// TwinCAT 3 PLC project TcoDrivesBeckhoff
// Title: TcoDrivesBeckhoff
// Company: Vortex.Library
// Author: TcOpenGroup
// ProjectVersion: 0.6.0.913
// ProgramVersion: 3.1.4024.12
// libraries:
//   Tc2_MC2, * (Beckhoff Automation GmbH)
//   Tc2_MC2_Drive, * (Beckhoff Automation GmbH)
//   Tc2_Standard, * (Beckhoff Automation GmbH)
//   Tc2_System, * (Beckhoff Automation GmbH)
//   Tc3_Module, * (Beckhoff Automation GmbH)
//   TcoCore, 0.6.0.913 (Vortex.Library)
// project tree:
//   DUTs/ eAxisParameter.TcDUT, eAxisEncoderReferenceSystem.TcDUT, eDirection.TcDUT, eAxisStates.TcDUT, eEncoderReferenceMode.TcDUT, eHomingMode.TcDUT, ePowerOverride.TcDUT, eSetPositionMode.TcDUT, eJogMode.TcDUT, TcoAxisOpModes.TcDUT, TcoAxisRef.TcPOU, TcoAxisStatus.TcDUT, TcoAxisConfig.TcDUT
//   / PlcTask.TcTTO (not stored)
//   POUs/Conversions/ Tc2MC2_TO_Tco_AxisStates.TcPOU, LREAL_TO_Tco_AxisEncoderReferenceSystem.TcPOU, Tc2MC2_TO_Tco_SetPositionMode.TcPOU, Tc2MC2_TO_Tco_JogMode.TcPOU, Tco_TO_Tc2MC2_SetPositionMode.TcPOU, Tco_TO_Tc2MC2_Direction.TcPOU, Tc2MC2_TO_Tco_Direction.TcPOU, Tco_TO_Tc2MC2_HomingMode.TcPOU, Tco_TO_Tc2MC2_EncRefMode.TcPOU, Tc2MC2_TO_Tco_EncRefMode.TcPOU, Tc2MC2_TO_Tco_HomingMode.TcPOU, Tco_TO_Tc2MC2_AxisStates.TcPOU, Tco_TO_Tc2MC2_JogMode.TcPOU
//   POUs/ MAIN.TcPOU
//   POUs/Prototypes/CartesianCoordinateSystem/MultiAxisSystem/ eTcoMultiAxisSystem.TcDUT, ITcoMultiAxis.TcIO, TcoMultiAxis.TcPOU, TcoMultiAxisConfig.TcDUT, TcoMultiAxisStatus.TcDUT, TcoMultiAxisMoveParam.TcDUT, TcoMultiAxisPositionsRootContainer.TcPOU
//   POUs/Prototypes/CartesianCoordinateSystem/SingleAxisSystem/ ITcoSingleAxis.TcIO, TcoSingleAxisStatus.TcDUT, TcoSingleAxisConfig.TcDUT, TcoSingleAxis.TcPOU, TcoSingleAxisMoveParam.TcDUT, TcoSingleAxisPositionsRootContainer.TcPOU
//   POUs/Prototypes/CartesianCoordinateSystem/ TcoAxisExchangeDataTask.TcPOU
//   POUs/Prototypes/TcoDriveSimple/DriveState/ eTcoMovementState.TcDUT, TcoMovementState.TcPOU
//   POUs/Prototypes/TcoDriveSimple/ ITcoDriveSimple.TcIO, Power.TcPOU, Jog.TcPOU, TcoDriveSimple.TcPOU
//   POUs/Prototypes/TcoDriveSimple/MotionTasks/ HomeTask.TcPOU, MoveModuloTask.TcPOU, MoveRelativeTask.TcPOU, MoveAbsoluteTask.TcPOU, MoveVelocityTask.TcPOU, SetTorqueTask.TcPOU, StopTask.TcPOU, HaltTask.TcPOU
//   POUs/Prototypes/TcoDriveSimple/AxisTasks/ ResetTask.TcPOU, SetPositionTask.TcPOU, SoEResetTask.TcPOU
// real-time tasks:
//   TASK PlcTask: cycle T#10ms, priority 20, ADS port 350
//   TASK PlcTask1: cycle T#10ms, priority 1, ADS port 351
// motion (NC):
//   TASK NC-Task 1 SAF: cycle T#2ms, priority 4, ADS port 501
//   TASK NC-Task 1 SVB: cycle T#10ms, priority 8, ADS port 511
//   AXIS Axis 1 (id 1)
//     Dynamic: Acceleration=5979.5, Deceleration=5979.5, Jerk=17938.5
//     Velo: RefSearch=39.8633642666667, RefSync=39.8633642666667, SlowManual=199.316821333333, FastManual=1195.900928, Fast=3986.33642666667, Maximum=3986.34
//     OtherSettings: AllowMotionCmdToSlave=true
//     encoder EncType=1
//       EncPara: ScaleFactorNumerator=104.8576, ScaleFactorDenominator=1048576, Offset=-0.001200000000608
//     drive DrvType=5
//       Analog: VeloReferenz=4384.97006933333, TorqueSetpointScale=10, ScaleFactorActTorque=0.1
//       TimeComp: TaskDelayCycles=1
//     controller CtrType=1
//       CtrPara: PriorControlFactor=1
//         Observer: BandWidth=20
//   AXIS Axis 2 (id 2)
//     Dynamic: Acceleration=500, Deceleration=500, Jerk=1000
//     Velo: SlowManual=10, FastManual=50, Maximum=3986.34
//     OtherSettings: AllowMotionCmdToSlave=true
//     encoder EncType=1
//       EncPara: ScaleFactorNumerator=1, ScaleFactorDenominator=1024
//     drive DrvType=5
//       Analog: VeloReferenz=4384.97006933333, TorqueSetpointScale=10, ScaleFactorActTorque=0.1
//       TimeComp: TaskDelayCycles=1
//     controller CtrType=1
//       CtrPara: PriorControlFactor=1
//         PosDiffControl: Enable=false
//         PID: PosKp=0.1
//         Observer: BandWidth=20
//   AXIS Axis 3 (id 3)
//     Dynamic: Acceleration=500, Deceleration=500, Jerk=1000
//     Velo: SlowManual=10, FastManual=50, Maximum=3986.34
//     OtherSettings: AllowMotionCmdToSlave=true
//     encoder EncType=1
//       EncPara: ScaleFactorNumerator=1, ScaleFactorDenominator=1024
//     drive DrvType=5
//       Analog: VeloReferenz=4384.97006933333, TorqueSetpointScale=10, ScaleFactorActTorque=0.1
//       TimeComp: TaskDelayCycles=1
//     controller CtrType=1
//       CtrPara: PriorControlFactor=1
//         PosDiffControl: Enable=false
//         PID: PosKp=0.1
//         Observer: BandWidth=20
//   AXIS Axis 4 (id 4)
//     Dynamic: Acceleration=500, Deceleration=500, Jerk=1000
//     Velo: SlowManual=10, FastManual=50, Maximum=3986.34
//     OtherSettings: AllowMotionCmdToSlave=true
//     encoder EncType=1
//       EncPara: ScaleFactorNumerator=1, ScaleFactorDenominator=1024
//     drive DrvType=5
//       Analog: VeloReferenz=4384.97006933333, TorqueSetpointScale=10, ScaleFactorActTorque=0.1
//       TimeComp: TaskDelayCycles=1
//     controller CtrType=1
//       CtrPara: PriorControlFactor=1
//         PosDiffControl: Enable=false
//         PID: PosKp=0.1
//         Observer: BandWidth=20
// I/O:
//   DEVICE Device 4 (EtherCAT) (disabled), AmsNetId 172.20.10.104.5.1
//     Term 1 (EK1100) [EK1100 EtherCAT Coupler (2A E-Bus)]
//       Term 2 (EL1008) [EL1008 8Ch. Dig. Input 24V, 3ms]
//       Term 3 (EL2008) [EL2008 8Ch. Dig. Output 24V, 0.5A]
//       Term 4 (EL3052) [EL3052 2Ch. Ana. Input 4-20mA]
//       Term 5 (EL9576) [EL9576 Brake chopper terminal]
//       Term 6 (EL7211-0010) [EL7211-0010 1Ch. MDP742 Servo motor output stage with OCT (50V, 4.5A RMS)]
//       Term 14 (EL7047) [EL7047 1Ch. Stepper motor output stage (50V, 5A)]
//       Term 8 (EL9011) [EL9011 End Terminal]
//   DEVICE Device 1 (EtherCAT) (disabled), AmsNetId 192.168.4.1.2.1
//     Drive 7 (IndraDrive MPB20) [IndraDrive MPB20]
//   DEVICE Device 2 (EtherCAT) (disabled), AmsNetId 192.168.4.1.3.1
//     Term 1 (EK1200) [EK1200-5000 EtherCAT Power supply (2A E-Bus)]
//       Term 10 (EK1122) [EK1122 2 port EtherCAT junction]
//       Term 11 (EL6002) [EL6002 Interface 2Ch. (RS232)]
//       Term 12 (EL1809) [EL1809 16Ch. Dig. Input 24V, 3ms]
//       Term 13 (EL2809) [EL2809 16Ch. Dig. Output 24V, 0.5A]
//       Term 15 (EL4004) [EL4004 4Ch. Ana. Output 0-10V, 12bit]
//       Term 16 (EL7342) [EL7342 2Ch. DC motor output stage (50V, 3.5A)]
//       Term 17 (EL4004) [EL4004 4Ch. Ana. Output 0-10V, 12bit]
//       Term 18 (EL6001) [EL6001 Interface (RS232)]
//       Term 10 (EL9011) [EL9011 End Terminal]
// variable links:
//   TcoDrivesBeckhoffTests/TcoDrivesBeckhoffTests Instance <-> Device 2 (EtherCAT)/Term 1 (EK1200)/Term 12 (EL1809)
//     PlcTask1 Inputs/GVL._calibrationCam <-> Channel 1/Input
//   TcoDrivesBeckhoffTests/TcoDrivesBeckhoffTests Instance <-> NC-Task 1 SAF/Axes/Axis 1
//     PlcTask1 Inputs/GVL.Axis1.NcToPlc <-> Outputs/ToPlc
//     PlcTask1 Outputs/GVL.Axis1.PlcToNc <-> Inputs/FromPlc
//   TcoDrivesBeckhoffTests/TcoDrivesBeckhoffTests Instance <-> NC-Task 1 SAF/Axes/Axis 2
//     PlcTask1 Inputs/GVL.Axis2.NcToPlc <-> Outputs/ToPlc
//     PlcTask1 Outputs/GVL.Axis2.PlcToNc <-> Inputs/FromPlc
//   TcoDrivesBeckhoffTests/TcoDrivesBeckhoffTests Instance <-> NC-Task 1 SAF/Axes/Axis 3
//     PlcTask1 Inputs/GVL.Axis3.NcToPlc <-> Outputs/ToPlc
//     PlcTask1 Outputs/GVL.Axis3.PlcToNc <-> Inputs/FromPlc
//   TcoDrivesBeckhoffTests/TcoDrivesBeckhoffTests Instance <-> NC-Task 1 SAF/Axes/Axis 4
//     PlcTask1 Inputs/GVL.Axis4.NcToPlc <-> Outputs/ToPlc
//     PlcTask1 Outputs/GVL.Axis4.PlcToNc <-> Inputs/FromPlc

// ---- DUTs/eAxisParameter.TcDUT
{attribute 'qualified_only'}
{attribute 'strict'}
TYPE eAxisParameter :
(
    (* PLCopen specific parameters *) (* Index-Group 0x4000 + ID*)
    CommandedPosition := 1, (* lreal *) (* taken from NcToPlc *)
    SWLimitPos, (* lreal *) (* IndexOffset= 16#0001_000E *)
    SWLimitNeg, (* lreal *) (* IndexOffset= 16#0001_000D *)
    EnableLimitPos, (* bool  *) (* IndexOffset= 16#0001_000C *)
    EnableLimitNeg, (* bool  *) (* IndexOffset= 16#0001_000B *)
    EnablePosLagMonitoring, (* bool  *) (* IndexOffset= 16#0002_0010 *)
    MaxPositionLag, (* lreal *) (* IndexOffset= 16#0002_0012 *)
    MaxVelocitySystem, (* lreal *) (* IndexOffset= 16#0000_0027 *)
    MaxVelocityAppl, (* lreal *) (* IndexOffset= 16#0000_0027 *)
    ActualVelocity, (* lreal *) (* taken from NcToPlc *)
    CommandedVelocity, (* lreal *) (* taken from NcToPlc *)
    MaxAccelerationSystem, (* lreal *) (* IndexOffset= 16#0000_0101 *)
    MaxAccelerationAppl, (* lreal *) (* IndexOffset= 16#0000_0101 *)
    MaxDecelerationSystem, (* lreal *) (* IndexOffset= 16#0000_0102 *)
    MaxDecelerationAppl, (* lreal *) (* IndexOffset= 16#0000_0102 *)
    MaxJerkSystem, (* lreal *) (* IndexOffset= 16#0000_0103 *)
    MaxJerkAppl, (* lreal *) (* IndexOffset= 16#0000_0103 *)
    (* Beckhoff specific parameters *) (* Index-Group 0x4000 + ID*)
    AxisId := 1000, (* lreal *) (* IndexOffset= 16#0000_0001 *)
    AxisVeloManSlow, (* lreal *) (* IndexOffset= 16#0000_0008 *)
    AxisVeloManFast, (* lreal *) (* IndexOffset= 16#0000_0009 *)
    AxisVeloMax, (* lreal *) (* IndexOffset= 16#0000_0027 *)
    AxisAcc, (* lreal *) (* IndexOffset= 16#0000_0101 *)
    AxisDec, (* lreal *) (* IndexOffset= 16#0000_0102 *)
    AxisJerk, (* lreal *) (* IndexOffset= 16#0000_0103 *)
    MaxJerk, (* lreal *) (* IndexOffset= 16#0000_0103 *)
    AxisMaxVelocity, (* lreal *) (* IndexOffset= 16#0000_0027 *)
    AxisRapidTraverseVelocity, (* lreal *) (* IndexOffset= 16#0000_000A *)
    AxisManualVelocityFast, (* lreal *) (* IndexOffset= 16#0000_0009 *)
    AxisManualVelocitySlow, (* lreal *) (* IndexOffset= 16#0000_0008 *)
    AxisCalibrationVelocityForward, (* lreal *) (* IndexOffset= 16#0000_0006 *)
    AxisCalibrationVelocityBackward, (* lreal *) (* IndexOffset= 16#0000_0007 *)
    AxisJogIncrementForward, (* lreal *) (* IndexOffset= 16#0000_0018 *)
    AxisJogIncrementBackward, (* lreal *) (* IndexOffset= 16#0000_0019 *)
    AxisEnMinSoftPosLimit, (* bool  *) (* IndexOffset= 16#0001_000B *)
    AxisMinSoftPosLimit, (* lreal *) (* IndexOffset= 16#0001_000D *)
    AxisEnMaxSoftPosLimit, (* bool  *) (* IndexOffset= 16#0001_000C *)
    AxisMaxSoftPosLimit, (* lreal *) (* IndexOffset= 16#0001_000E *)
    AxisEnPositionLagMonitoring, (* bool  *) (* IndexOffset= 16#0002_0010 *)
    AxisMaxPosLagValue, (* lreal *) (* IndexOffset= 16#0002_0012 *)
    AxisMaxPosLagFilterTime, (* lreal *) (* IndexOffset= 16#0002_0013 *)
    AxisEnPositionRangeMonitoring, (* bool  *) (* IndexOffset= 16#0000_000F *)
    AxisPositionRangeWindow, (* lreal *) (* IndexOffset= 16#0000_0010 *)
    AxisEnTargetPositionMonitoring, (* bool  *) (* IndexOffset= 16#0000_0015 *)
    AxisTargetPositionWindow, (* lreal *) (* IndexOffset= 16#0000_0016 *)
    AxisTargetPositionMonitoringTime, (* lreal *) (* IndexOffset= 16#0000_0017 *)
    AxisEnInTargetTimeout, (* bool  *) (* IndexOffset= 16#0000_0029 *)
    AxisInTargetTimeout, (* lreal *) (* IndexOffset= 16#0000_002A *)
    AxisEnMotionMonitoring, (* bool  *) (* IndexOffset= 16#0000_0011 *)
    AxisMotionMonitoringWindow, (* lreal *) (* IndexOffset= 16#0000_0028 *)
    AxisMotionMonitoringTime, (* lreal *) (* IndexOffset= 16#0000_0012 *)
    AxisDelayTimeVeloPosition, (* lreal *) (* IndexOffset= 16#0000_0104 *)
    AxisEnLoopingDistance, (* bool  *) (* IndexOffset= 16#0000_0013 *)
    AxisLoopingDistance, (* lreal *) (* IndexOffset= 16#0000_0014 *)
    AxisEnBacklashCompensation, (* bool  *) (* IndexOffset= 16#0000_002B *)
    AxisBacklash, (* lreal *) (* IndexOffset= 16#0000_002C *)
    AxisEnDataPersistence, (* bool  *) (* IndexOffset= 16#0000_0030 *)
    AxisRefVeloOnRefOutput, (* lreal *) (* IndexOffset= 16#0003_0101 *)
    AxisOverrideType, (* lreal *) (* IndexOffset= 16#0000_0105 *)
    (* new since 4/2007 *)
    AxisEncoderScalingFactor, (* lreal *) (* IndexOffset= 16#0001_0006 *)
    AxisEncoderOffset, (* lreal *) (* IndexOffset= 16#0001_0007 *)
    AxisEncoderDirectionInverse, (* bool  *) (* IndexOffset= 16#0001_0008 *)
    AxisEncoderMask, (* dword *) (* IndexOffset= 16#0001_0015 *)
    AxisEncoderModuloValue, (* lreal *) (* IndexOffset= 16#0001_0009 *)
    AxisModuloToleranceWindow, (* lreal *) (* IndexOffset= 16#0001_001B *)
    AxisEnablePosCorrection, (* bool  *) (* IndexOffset= 16#0001_0016 *)
    AxisPosCorrectionFilterTime, (* lreal *) (* IndexOffset= 16#0001_0017 *)
    (* new since 1/2010 *)
    AxisUnitInterpretation, (* lreal *) (* IndexOffset= 16#0000_0026 *)
    AxisMotorDirectionInverse, (* bool  *) (* IndexOffset= 16#0003_0006 *)
    (* new since 1/2011 *)
    AxisCycleTime, (* lreal *) (* IndexOffset= 16#0000_0004 *)
    (* new since 5/2011 *)
    AxisFastStopSignalType, (* dword *) (* IndexOffset= 16#0000_001E *)
    AxisFastAcc, (* lreal *) (* IndexOffset= 16#0000_010A *)
    AxisFastDec, (* lreal *) (* IndexOffset= 16#0000_010B *)
    AxisFastJerk, (* lreal *) (* IndexOffset= 16#0000_010C *)
    (* new since 1/2012 *)
    AxisEncoderScalingNumerator, (* lreal *) (* IndexOffset= 16#0001_0023 - available in Tc3 *)
    AxisEncoderScalingDenominator, (* lreal *) (* IndexOffset= 16#0001_0024 - available in Tc3 *)
    (* new since 7/2016 *)
    AxisMaximumAcceleration, (* lreal *) (* IndexOffset= 16#0000_00F1 - available in Tc3 *)
    AxisMaximumDeceleration, (* lreal *) (* IndexOffset= 16#0000_00F2 - available in Tc3 *)
    AxisVeloJumpFactor, (* lreal *) (* IndexOffset= 16#0000_0106 *)
    AxisToleranceBallAuxAxis, (* lreal *) (* IndexOffset= 16#0000_0108 *)
    AxisMaxPositionDeviationAuxAxis, (* lreal *) (* IndexOffset= 16#0000_0109 *)
    AxisErrorPropagationMode, (* dword *) (* IndexOffset= 16#0000_001A *)
    AxisErrorPropagationDelay, (* lreal *) (* IndexOffset= 16#0000_001B *)
    AxisCoupleSlaveToActualValues, (* bool  *) (* IndexOffset= 16#0000_001C *)
    AxisAllowMotionCmdToSlaveAxis, (* bool  *) (* IndexOffset= 16#0000_0020 *)
    AxisAllowMotionCmdToExtSetAxis, (* bool  *) (* IndexOffset= 16#0000_0021 *)
    AxisEncoderSubMask, (* dword *) (* IndexOffset= 16#0001_0108 *)
    AxisEncoderReferenceSystem, (* dword *) (* IndexOffset= 16#0001_0019 *)
    AxisEncoderPositionFilterPT1, (* lreal *) (* IndexOffset= 16#0001_0010 *)
    AxisEncoderVelocityFilterPT1, (* lreal *) (* IndexOffset= 16#0001_0011 *)
    AxisEncoderAccelerationFilterPT1, (* lreal *) (* IndexOffset= 16#0001_0012 *)
    AxisEncoderMode, (* dword *) (* IndexOffset= 16#0001_000A *)
    AxisEncoderHomingInvDirCamSearch, (* bool  *) (* IndexOffset= 16#0001_0101 *)
    AxisEncoderHomingInvDirSyncSearch, (* bool  *) (* IndexOffset= 16#0001_0102 *)
    AxisEncoderHomingCalibValue, (* lreal *) (* IndexOffset= 16#0001_0103 *)
    AxisEncoderReferenceMode, (* dword *) (* IndexOffset= 16#0001_0107 *)
    AxisRefVeloOutputRatio, (* lreal *) (* IndexOffset= 16#0003_0102 *)
    AxisDrivePositionOutputScaling, (* lreal *) (* IndexOffset= 16#0003_0109 *)
    AxisDriveVelocityOutputScaling, (* lreal *) (* IndexOffset= 16#0003_0105 *)
    AxisDriveVelocityOutputDelay, (* lreal *) (* IndexOffset= 16#0003_010D *)
    AxisDriveMinOutputLimitation, (* lreal *) (* IndexOffset= 16#0003_000B *)
    AxisDriveMaxOutputLimitation, (* lreal *) (* IndexOffset= 16#0003_000C *)
    AxisTorqueInputScaling, (* lreal *) (* IndexOffset= 16#0003_0031 - available in Tc3 *)
    AxisTorqueInputFilterPT1, (* lreal *) (* IndexOffset= 16#0003_0032 - available in Tc3 *)
    AxisTorqueDerivationInputFilterPT1, (* lreal *) (* IndexOffset= 16#0003_0033 - available in Tc3 *)
    AxisTorqueOutputScaling, (* lreal *) (* IndexOffset= 16#0003_010B *)
    AxisTorqueOutputDelay, (* lreal *) (* IndexOffset= 16#0003_010F *)
    AxisAccelerationOutputScaling, (* lreal *) (* IndexOffset= 16#0003_010A *)
    AxisAccelerationOutputDelay, (* lreal *) (* IndexOffset= 16#0003_010E *)
    AxisDrivePosOutputSmoothFilterType, (* dword *) (* IndexOffset= 16#0003_0110 *)
    AxisDrivePosOutputSmoothFilterTime, (* lreal *) (* IndexOffset= 16#0003_0111 *)
    AxisDrivePosOutputSmoothFilterOrder, (* dword *) (* IndexOffset= 16#0003_0112 *)
    AxisDriveMode, (* dword *) (* IndexOffset= 16#0003_000A *)
    AxisDriftCompensationOffset, (* lreal *) (* IndexOffset= 16#0003_0104 *)
    AxisPositionControlKv, (* lreal *) (* IndexOffset= 16#0002_0102 *)
    AxisCtrlVelocityPreCtrlWeight, (* lreal *) (* IndexOffset= 16#0002_000B *)
    AxisControllerMode, (* dword *) (* IndexOffset= 16#0002_000A *)
    AxisCtrlAutoOffset, (* bool  *) (* IndexOffset= 16#0002_0110 *)
    AxisCtrlAutoOffsetTimer, (* lreal *) (* IndexOffset= 16#0002_0115 *)
    AxisCtrlAutoOffsetLimit, (* lreal *) (* IndexOffset= 16#0002_0114 *)
    AxisSlaveCouplingControlKcp, (* lreal *) (* IndexOffset= 16#0002_010F *)
    AxisCtrlOutputLimit, (* lreal *) (* IndexOffset= 16#0002_0100 *)
    (* Beckhoff specific axis status information - READ ONLY *) (* Index-Group 0x4100 + ID*)
    AxisTargetPosition := 2000, (* lreal *) (* IndexOffset= 16#0000_0013 *)
    AxisRemainingTimeToGo, (* lreal *) (* IndexOffset= 16#0000_0014 *)
    AxisRemainingDistanceToGo, (* lreal *) (* IndexOffset= 16#0000_0022, 16#0000_0042 *)
    (* Beckhoff specific axis functions *)
    (* read/write gear ratio of a slave *)
    AxisGearRatio := 3000, (* lreal *) (* read: IndexGroup=0x4100+ID, IdxOffset=16#0000_0022, *)
    (* write:IndexGroup=0x4200+ID, IdxOffset=16#0000_0042 *)
    (* Beckhoff specific other parameters *)
    (* new since 1/2011 *)
    NcSafCycleTime := 4000, (* lreal *) (* IndexOffset= 16#0000_0010 *)
    NcSvbCycleTime (* lreal *) (* IndexOffset= 16#0000_0012 *)
);
END_TYPE

// ---- DUTs/eAxisEncoderReferenceSystem.TcDUT
{attribute 'qualified_only'}
{attribute 'strict'}
TYPE eAxisEncoderReferenceSystem :
(
    INCREMENTAL := 0,
    ABSOLUTE := 1,
    ABSOLUTE_MODULO := 2,
    ABSOLUTE_MULTITURN := 3,
    INCREMENTAL_SINGLETURN_ABSOLUTE := 4,
    ABSOLUTE_SINGLETURN := 5
);
END_TYPE

// ---- DUTs/eDirection.TcDUT
TYPE eDirection :
(
    MC_Positive_Direction := 1,
    MC_Shortest_Way := 2,
    MC_Negative_Direction := 3,
    MC_Current_Direction := 4,
    MC_Undefined_Direction := 128
) INT;
END_TYPE

// ---- DUTs/eAxisStates.TcDUT
TYPE eAxisStates :
(
    MC_AXISSTATE_UNDEFINED := 0,
    MC_AXISSTATE_DISABLED := 1,
    MC_AXISSTATE_STANDSTILL := 2,
    MC_AXISSTATE_ERRORSTOP := 3,
    MC_AXISSTATE_STOPPING := 4,
    MC_AXISSTATE_HOMING := 5,
    MC_AXISSTATE_DISCRETEMOTION := 6,
    MC_AXISSTATE_CONTINOUSMOTION := 7,
    MC_AXISSTATE_SYNCHRONIZEDMOTION := 8
);
END_TYPE

// ---- DUTs/eEncoderReferenceMode.TcDUT
TYPE eEncoderReferenceMode :
(
    ENCODERREFERENCEMODE_DEFAULT := 0,
    ENCODERREFERENCEMODE_PLCCAM := 1,
    ENCODERREFERENCEMODE_HARDWARESYNC := 2,
    ENCODERREFERENCEMODE_HARDWARELATCHPOS := 3,
    ENCODERREFERENCEMODE_HARDWARELATCHNEG := 4,
    ENCODERREFERENCEMODE_SOFTWARESYNC := 5,
    ENCODERREFERENCEMODE_SOFTDRIVELATCHPOS := 6,
    ENCODERREFERENCEMODE_SOFTDRIVELATCHNEG := 7
) UDINT;
END_TYPE

// ---- DUTs/eHomingMode.TcDUT
TYPE eHomingMode :
(
    MC_DefaultHoming := 0,
    MC_Direct := 4,
    MC_ForceCalibration := 7,
    MC_ResetCalibration := 8
) INT;
END_TYPE

// ---- DUTs/ePowerOverride.TcDUT
{attribute 'qualified_only'}
{attribute 'strict'}
TYPE ePowerOverride :
(
    Global_control := 0,
    Local_control := 1
);
END_TYPE

// ---- DUTs/eSetPositionMode.TcDUT
{attribute 'qualified_only'}
{attribute 'strict'}
TYPE eSetPositionMode :
(
    Absolute := 0,
    Relative := 1
);
END_TYPE

// ---- DUTs/eJogMode.TcDUT
{attribute 'qualified_only'}
{attribute 'strict'}
TYPE eJogMode :
(
    MC_JOGMODE_STANDARD_SLOW, (* motion with standard jog parameters for slow motion *)
    MC_JOGMODE_STANDARD_FAST, (* motion with standard jog parameters for fast motion *)
    MC_JOGMODE_CONTINOUS, (* axis moves as long as the jog button is pressed using parameterized dynamics *)
    MC_JOGMODE_INCHING, (* axis moves for a certain relative distance *)
    MC_JOGMODE_INCHING_MODULO (* axis moves for a certain relative distance - stop position is rounded to the distance value *)
);
END_TYPE

// ---- DUTs/TcoAxisOpModes.TcDUT
TYPE TcoAxisOpModes :
STRUCT
    PositionAreaMonitoring : BOOL; (* bit 0 - OpModeDWord *)
    TargetPositionMonitoring : BOOL; (* bit 1 - OpModeDWord *)
    LoopMode : BOOL; (* bit 2 - OpModeDWord - loop mode for two speed axes *)
    MotionMonitoring : BOOL; (* bit 3 - OpModeDWord *)
    PEHTimeMonitoring : BOOL; (* bit 4 - OpModeDWord *)
    BacklashCompensation : BOOL; (* bit 5 - OpModeDWord *)
    Modulo : BOOL; (* bit 7 - OpModeDWord - axis is parameterized as modulo axis *)
    PositionLagMonitoring : BOOL; (* bit 16 - OpModeDWord *)
    VelocityLagMonitoring : BOOL; (* bit 17 - OpModeDWord *)
    SoftLimitMinMonitoring : BOOL; (* bit 18 - OpModeDWord *)
    SoftLimitMaxMonitoring : BOOL; (* bit 19 - OpModeDWord *)
    PositionCorrection : BOOL; (* bit 20 - OpModeDWord *)
END_STRUCT
END_TYPE

// ---- DUTs/TcoAxisStatus.TcDUT
TYPE TcoAxisStatus :
STRUCT
    {attribute addProperty Name "<#Actual position#>"}
    ActPos : LREAL; (* Actual position (absolut value from NC) *)
    {attribute addProperty Name "<#Actual modulo position#>"}
    ModuloActPos : LREAL; (* Actual modulo position *)
    {attribute addProperty Name "<#Actual modulo turns#>"}
    ModuloActTurns : DINT; (* Actual modulo turns *)
    {attribute addProperty Name "<#Actual velocity#>"}
    ActVelo : LREAL; (* Actual velocity *)
    {attribute addProperty Name "<#Actual acceleration#>"}
    ActAcc : LREAL;
    {attribute addProperty Name "<#Actual torque#>"}
    ActTorque : LREAL;
    {attribute addProperty Name "<#Command number#>"}
    CmdNo : WORD; (* Continuous actual command number *)
    {attribute addProperty Name "<#Command state#>"}
    CmdState : WORD; (* Command state *)
    {attribute addProperty Name "<#Motion state#>"}
    MotionState : eAxisStates; (* motion state in the PLCopen state diagram *)
    {attribute addProperty Name "<#Error#>"}
    Error : BOOL; (* axis error state *)
    {attribute addProperty Name "<#Error id#>"}
    ErrorId : UDINT; (* axis error code *)
    (* PLCopen motion control statemachine states: *)
    ErrorStop : BOOL;
    Disabled : BOOL;
    Stopping : BOOL;
    StandStill : BOOL;
    DiscreteMotion : BOOL;
    ContinuousMotion : BOOL;
    SynchronizedMotion : BOOL;
    Homing : BOOL;
    (* additional status - (PLCopen definition)*)
    ConstantVelocity : BOOL;
    Accelerating : BOOL;
    Decelerating : BOOL;
    (* Axis.NcToPlc.StateDWord *)
    Operational : BOOL;
    ControlLoopClosed : BOOL; (* operational and position control active *)
    HasJob : BOOL;
    HasBeenStopped : BOOL;
    NewTargetPosition : BOOL; (* new target position commanded during move *)
    InPositionArea : BOOL;
    InTargetPosition : BOOL;
    Homed : BOOL;
    HomingBusy : BOOL;
    MotionCommandsLocked : BOOL; (* stop 'n hold *)
    SoftLimitMinExceeded : BOOL; (* reverse soft travel limit exceeded *)
    SoftLimitMaxExceeded : BOOL; (* forward soft travel limit exceeded *)
    Moving : BOOL;
    PositiveDirection : BOOL;
    NegativeDirection : BOOL;
    NotMoving : BOOL;
    Compensating : BOOL; (* superposition - overlayed motion *)
    ExtSetPointGenEnabled : BOOL;
    ExternalLatchValid : BOOL;
    CamDataQueued : BOOL;
    CamTableQueued : BOOL;
    CamScalingPending : BOOL;
    CmdBuffered : BOOL;
    PTPmode : BOOL;
    DriveDeviceError : BOOL;
    IoDataInvalid : BOOL;
    (* Axis.NcToPlc.CoupleState *)
    Coupled : BOOL;
    (* axis operation mode feedback from NcToPlc *)
    OpMode : TcoAxisOpModes;
END_STRUCT
END_TYPE

// ---- DUTs/TcoAxisConfig.TcDUT
TYPE TcoAxisConfig :
STRUCT
    {attribute addProperty Name "<#Hide Power Tab#>"}
    HidePower : BOOL;
    {attribute addProperty Name "<#Hide Reset Tab#>"}
    HideReset : BOOL;
    {attribute addProperty Name "<#Hide Stop Tab#>"}
    HideStop : BOOL;
    {attribute addProperty Name "<#Hide Halt Tab#>"}
    HideHalt : BOOL;
    {attribute addProperty Name "<#Hide Homing Tab#>"}
    HideHoming : BOOL;
    {attribute addProperty Name "<#Hide Jogging Tab#>"}
    HideJogging : BOOL;
    {attribute addProperty Name "<#Hide MoveRelative Tab#>"}
    HideMoveRelative : BOOL;
    {attribute addProperty Name "<#Hide MoveAbsolute Tab#>"}
    HideMoveAbsolute : BOOL;
    {attribute addProperty Name "<#Hide MoveModulo Tab#>"}
    HideMoveModulo : BOOL;
    {attribute addProperty Name "<#Hide MoveVelocity Tab#>"}
    HideMoveVelocity : BOOL;
    {attribute addProperty Name "<#Hide SetTorque Tab#>"}
    HideSetTorque : BOOL;
    {attribute addProperty Name "<#Override velocity in service [%]#>"}
    OverrideInService : LREAL;
END_STRUCT
END_TYPE

// ---- POUs/Prototypes/CartesianCoordinateSystem/MultiAxisSystem/eTcoMultiAxisSystem.TcDUT
{attribute 'qualified_only'}
{attribute 'strict'}
TYPE eTcoMultiAxisSystem :
(
    SingleAxisSystem := 1,
    TwoAxisSystem := 2,
    ThreeAxisSystem := 3,
    FourAxissystem := 4
);
END_TYPE

// ---- POUs/Prototypes/CartesianCoordinateSystem/MultiAxisSystem/TcoMultiAxisConfig.TcDUT
TYPE TcoMultiAxisConfig :
STRUCT
    Axis1Disabled : BOOL;
    Axis2Disabled : BOOL;
    Axis3Disabled : BOOL;
    Axis4Disabled : BOOL;
    InfoTime : TIME := T#2S;
    ErrorTime : TIME := T#5S;
    {attribute addProperty Name "<#Hide Load position Tab#>"}
    HideLoadPositionTask : BOOL;
    {attribute addProperty Name "<#Hide Save position Tab#>"}
    HideSavePositionTask : BOOL;
    {attribute addProperty Name "<#Hide MoveAbsolute Tab#>"}
    HideMoveAbsoluteTask : BOOL;
    {attribute addProperty Name "<#Hide Position Tab#>"}
    HidePositionTable : BOOL;
END_STRUCT
END_TYPE

// ---- POUs/Prototypes/CartesianCoordinateSystem/MultiAxisSystem/TcoMultiAxisStatus.TcDUT
TYPE TcoMultiAxisStatus :
STRUCT
    ActionDescription : STRING(100);
END_STRUCT
END_TYPE

// ---- POUs/Prototypes/CartesianCoordinateSystem/MultiAxisSystem/TcoMultiAxisMoveParam.TcDUT
TYPE TcoMultiAxisMoveParam :
STRUCT
    {attribute addProperty Name "<#Axis 1#>"}
    Axis1 : TcoSingleAxisMoveParam;
    {attribute addProperty Name "<#Axis 2#>"}
    Axis2 : TcoSingleAxisMoveParam;
    {attribute addProperty Name "<#Axis 3#>"}
    Axis3 : TcoSingleAxisMoveParam;
    {attribute addProperty Name "<#Axis 4#>"}
    Axis4 : TcoSingleAxisMoveParam;
END_STRUCT
END_TYPE

// ---- POUs/Prototypes/CartesianCoordinateSystem/SingleAxisSystem/TcoSingleAxisStatus.TcDUT
TYPE TcoSingleAxisStatus :
STRUCT
    ActionDescription : STRING(100);
END_STRUCT
END_TYPE

// ---- POUs/Prototypes/CartesianCoordinateSystem/SingleAxisSystem/TcoSingleAxisConfig.TcDUT
TYPE TcoSingleAxisConfig :
STRUCT
    InfoTime : TIME := T#2S;
    ErrorTime : TIME := T#5S;
    {attribute addProperty Name "<#Hide Load position Tab#>"}
    HideLoadPositionTask : BOOL;
    {attribute addProperty Name "<#Hide Save position Tab#>"}
    HideSavePositionTask : BOOL;
    {attribute addProperty Name "<#Hide MoveAbsolute Tab#>"}
    HideMoveAbsoluteTask : BOOL;
    {attribute addProperty Name "<#Hide MoveRelative Tab#>"}
    HideMoveRelativeTask : BOOL;
    {attribute addProperty Name "<#Hide Position Tab#>"}
    HidePositionTable : BOOL;
END_STRUCT
END_TYPE

// ---- POUs/Prototypes/CartesianCoordinateSystem/SingleAxisSystem/TcoSingleAxisMoveParam.TcDUT
TYPE TcoSingleAxisMoveParam :
STRUCT
    {attribute addProperty Name "<#Position#>"}
    Position : LREAL;
    {attribute addProperty Name "<#Velocity#>"}
    Velocity : LREAL;
    {attribute addProperty Name "<#Acceleration#>"}
    Acceleration : LREAL;
    {attribute addProperty Name "<#Deceleration#>"}
    Deceleration : LREAL;
    {attribute addProperty Name "<#Jerk#>"}
    Jerk : LREAL;
END_STRUCT
END_TYPE

// ---- POUs/Prototypes/TcoDriveSimple/DriveState/eTcoMovementState.TcDUT
{attribute 'qualified_only'}
{attribute 'strict'}
TYPE eTcoMovementState :
(
    WaitingForMovementTask := 0,
    Reset,
    Power,
    ParametersCheck,
    Movement,
    Error := 255
);
END_TYPE

// ---- POUs/Prototypes/CartesianCoordinateSystem/MultiAxisSystem/ITcoMultiAxis.TcIO
INTERFACE ITcoMultiAxis

METHOD MoveAbsolute : TcoCore.ITcoTaskStatus
VAR_INPUT
	MoveParams : TcoMultiAxisMoveParam;;
END_VAR
END_METHOD

PROPERTY MoveAbsoluteTask : REFERENCE TO TcoCore.TcoTask
GET
END_GET
END_PROPERTY

METHOD ResetDrives : TcoCore.ITcoTaskStatus
VAR_INPUT
END_VAR
END_METHOD

METHOD SoeReset : TcoCore.ITcoTaskStatus
VAR_INPUT
END_VAR
END_METHOD

END_INTERFACE

// ---- POUs/Prototypes/CartesianCoordinateSystem/SingleAxisSystem/ITcoSingleAxis.TcIO
INTERFACE ITcoSingleAxis

METHOD MoveAbsolute : TcoCore.ITcoTaskStatus
VAR_INPUT
	MoveParams : TcoSingleAxisMoveParam;
END_VAR
END_METHOD

PROPERTY PUBLIC MoveAbsoluteTask : REFERENCE TO TcoCore.TcoTask
GET
END_GET
END_PROPERTY

METHOD MoveRelative : TcoCore.ITcoTaskStatus
VAR_INPUT
	MoveParams : TcoSingleAxisMoveParam;
END_VAR
END_METHOD

PROPERTY PUBLIC MoveRelativeTask : REFERENCE TO TcoCore.TcoTask
GET
END_GET
END_PROPERTY

END_INTERFACE

// ---- POUs/Prototypes/TcoDriveSimple/ITcoDriveSimple.TcIO
INTERFACE ITcoDriveSimple

PROPERTY DriveRef : REFERENCE TO TcoDriveSimple
GET
END_GET
END_PROPERTY

END_INTERFACE

// ---- DUTs/TcoAxisRef.TcPOU
FUNCTION_BLOCK TcoAxisRef EXTENDS Tc2_MC2.AXIS_REF

END_FUNCTION_BLOCK

// ---- POUs/Conversions/Tc2MC2_TO_Tco_AxisStates.TcPOU
FUNCTION INTERNAL Tc2MC2_TO_Tco_AxisStates : BOOL
VAR_INPUT
    Tc2MC2AxisStates : Tc2_MC2.MC_AxisStates;
END_VAR
VAR_IN_OUT
    TcoAxisStates : eAxisStates;
END_VAR

CASE TcoAxisStates OF
    Tc2_MC2.MC_AxisStates.MC_AXISSTATE_CONTINOUSMOTION:
        TcoAxisStates := eAxisStates.MC_AXISSTATE_CONTINOUSMOTION;
        Tc2MC2_TO_Tco_AxisStates := TRUE;
    Tc2_MC2.MC_AxisStates.MC_AXISSTATE_DISABLED:
        TcoAxisStates := eAxisStates.MC_AXISSTATE_DISABLED;
        Tc2MC2_TO_Tco_AxisStates := TRUE;
    Tc2_MC2.MC_AxisStates.MC_AXISSTATE_DISCRETEMOTION:
        TcoAxisStates := eAxisStates.MC_AXISSTATE_DISCRETEMOTION;
        Tc2MC2_TO_Tco_AxisStates := TRUE;
    Tc2_MC2.MC_AxisStates.MC_AXISSTATE_ERRORSTOP:
        TcoAxisStates := eAxisStates.MC_AXISSTATE_ERRORSTOP;
        Tc2MC2_TO_Tco_AxisStates := TRUE;
    Tc2_MC2.MC_AxisStates.MC_AXISSTATE_HOMING:
        TcoAxisStates := eAxisStates.MC_AXISSTATE_HOMING;
        Tc2MC2_TO_Tco_AxisStates := TRUE;
    Tc2_MC2.MC_AxisStates.MC_AXISSTATE_STANDSTILL:
        TcoAxisStates := eAxisStates.MC_AXISSTATE_STANDSTILL;
        Tc2MC2_TO_Tco_AxisStates := TRUE;
    Tc2_MC2.MC_AxisStates.MC_AXISSTATE_STOPPING:
        TcoAxisStates := eAxisStates.MC_AXISSTATE_STOPPING;
        Tc2MC2_TO_Tco_AxisStates := TRUE;
    Tc2_MC2.MC_AxisStates.MC_AXISSTATE_SYNCHRONIZEDMOTION:
        TcoAxisStates := eAxisStates.MC_AXISSTATE_SYNCHRONIZEDMOTION;
        Tc2MC2_TO_Tco_AxisStates := TRUE;
    Tc2_MC2.MC_AxisStates.MC_AXISSTATE_UNDEFINED:
        TcoAxisStates := eAxisStates.MC_AXISSTATE_UNDEFINED;
        Tc2MC2_TO_Tco_AxisStates := TRUE;
ELSE
    Tc2MC2_TO_Tco_AxisStates := FALSE;
END_CASE

END_FUNCTION

// ---- POUs/Conversions/LREAL_TO_Tco_AxisEncoderReferenceSystem.TcPOU
FUNCTION INTERNAL LREAL_TO_Tco_AxisEncoderReferenceSystem : BOOL
VAR_INPUT
    inValue : LREAL;
END_VAR
VAR_IN_OUT
    TcoAxisEncoderReferenceSystem : eAxisEncoderReferenceSystem;
END_VAR
VAR
    _value : INT;
END_VAR

_value := LREAL_TO_INT(inValue);

CASE _value OF
    eAxisEncoderReferenceSystem.ABSOLUTE:
        TcoAxisEncoderReferenceSystem := eAxisEncoderReferenceSystem.ABSOLUTE;
        LREAL_TO_Tco_AxisEncoderReferenceSystem := TRUE;
    eAxisEncoderReferenceSystem.ABSOLUTE_MODULO:
        TcoAxisEncoderReferenceSystem := eAxisEncoderReferenceSystem.ABSOLUTE_MODULO;
        LREAL_TO_Tco_AxisEncoderReferenceSystem := TRUE;
    eAxisEncoderReferenceSystem.ABSOLUTE_MULTITURN:
        TcoAxisEncoderReferenceSystem := eAxisEncoderReferenceSystem.ABSOLUTE_MULTITURN;
        LREAL_TO_Tco_AxisEncoderReferenceSystem := TRUE;
    eAxisEncoderReferenceSystem.ABSOLUTE_SINGLETURN:
        TcoAxisEncoderReferenceSystem := eAxisEncoderReferenceSystem.ABSOLUTE_SINGLETURN;
        LREAL_TO_Tco_AxisEncoderReferenceSystem := TRUE;
    eAxisEncoderReferenceSystem.INCREMENTAL:
        TcoAxisEncoderReferenceSystem := eAxisEncoderReferenceSystem.INCREMENTAL;
        LREAL_TO_Tco_AxisEncoderReferenceSystem := TRUE;
    eAxisEncoderReferenceSystem.INCREMENTAL_SINGLETURN_ABSOLUTE:
        TcoAxisEncoderReferenceSystem := eAxisEncoderReferenceSystem.INCREMENTAL_SINGLETURN_ABSOLUTE;
        LREAL_TO_Tco_AxisEncoderReferenceSystem := TRUE;
ELSE
    LREAL_TO_Tco_AxisEncoderReferenceSystem := FALSE;
END_CASE

END_FUNCTION

// ---- POUs/Conversions/Tc2MC2_TO_Tco_SetPositionMode.TcPOU
FUNCTION INTERNAL Tc2MC2_TO_Tco_SetPositionMode : BOOL
VAR_INPUT
    Tc2MC2SetPositionMode : BOOL;
END_VAR
VAR_IN_OUT
    TcoSetPositionMode : eSetPositionMode;
END_VAR

IF Tc2MC2SetPositionMode THEN
    TcoSetPositionMode := eSetPositionMode.Absolute;
    Tc2MC2_TO_Tco_SetPositionMode := TRUE;
ELSE
    TcoSetPositionMode := eSetPositionMode.Relative;
    Tc2MC2_TO_Tco_SetPositionMode := TRUE;
END_IF

END_FUNCTION

// ---- POUs/Conversions/Tc2MC2_TO_Tco_JogMode.TcPOU
FUNCTION INTERNAL Tc2MC2_TO_Tco_JogMode : BOOL
VAR_INPUT
    Tc2MC2JogMode : Tc2_MC2.E_JogMode;
END_VAR
VAR_IN_OUT
    TcoJogMode : eJogMode;
END_VAR

CASE Tc2MC2JogMode OF
    Tc2_MC2.MC_JOGMODE_STANDARD_SLOW:
        TcoJogMode := eJogMode.MC_JOGMODE_STANDARD_SLOW;
        Tc2MC2_TO_Tco_JogMode := TRUE;
    Tc2_MC2.MC_JOGMODE_STANDARD_FAST:
        TcoJogMode := eJogMode.MC_JOGMODE_STANDARD_FAST;
        Tc2MC2_TO_Tco_JogMode := TRUE;
    Tc2_MC2.MC_JOGMODE_CONTINOUS:
        TcoJogMode := eJogMode.MC_JOGMODE_CONTINOUS;
        Tc2MC2_TO_Tco_JogMode := TRUE;
    Tc2_MC2.MC_JOGMODE_INCHING:
        TcoJogMode := eJogMode.MC_JOGMODE_INCHING;
        Tc2MC2_TO_Tco_JogMode := TRUE;
    Tc2_MC2.MC_JOGMODE_INCHING_MODULO:
        TcoJogMode := eJogMode.MC_JOGMODE_INCHING_MODULO;
        Tc2MC2_TO_Tco_JogMode := TRUE;
ELSE
    Tc2MC2_TO_Tco_JogMode := FALSE;
END_CASE

END_FUNCTION

// ---- POUs/Conversions/Tco_TO_Tc2MC2_SetPositionMode.TcPOU
FUNCTION INTERNAL Tco_TO_Tc2MC2_SetPositionMode : BOOL
VAR_INPUT
    TcoSetPositionMode : eSetPositionMode;
END_VAR
VAR_IN_OUT
    Tc2MC2SetPositionMode : BOOL;
END_VAR

CASE TcoSetPositionMode OF
    eSetPositionMode.Absolute:
        Tc2MC2SetPositionMode := TRUE;
        Tco_TO_Tc2MC2_SetPositionMode := TRUE;
    eSetPositionMode.Relative:
        Tc2MC2SetPositionMode := FALSE;
        Tco_TO_Tc2MC2_SetPositionMode := TRUE;
ELSE
    Tco_TO_Tc2MC2_SetPositionMode := FALSE;
END_CASE

END_FUNCTION

// ---- POUs/Conversions/Tco_TO_Tc2MC2_Direction.TcPOU
FUNCTION INTERNAL Tco_TO_Tc2MC2_Direction : BOOL
VAR_INPUT
    TcoDirection : eDirection;
END_VAR
VAR_IN_OUT
    Tc2MC2Direction : Tc2_MC2.MC_Direction;
END_VAR

CASE TcoDirection OF
    eDirection.MC_Current_Direction:
        Tc2MC2Direction := Tc2_MC2.MC_Direction.MC_Current_Direction;
        Tco_TO_Tc2MC2_Direction := TRUE;
    eDirection.MC_Negative_Direction:
        Tc2MC2Direction := Tc2_MC2.MC_Direction.MC_Negative_Direction;
        Tco_TO_Tc2MC2_Direction := TRUE;
    eDirection.MC_Positive_Direction:
        Tc2MC2Direction := Tc2_MC2.MC_Direction.MC_Positive_Direction;
        Tco_TO_Tc2MC2_Direction := TRUE;
    eDirection.MC_Shortest_Way:
        Tc2MC2Direction := Tc2_MC2.MC_Direction.MC_Shortest_Way;
        Tco_TO_Tc2MC2_Direction := TRUE;
    eDirection.MC_Undefined_Direction:
        Tc2MC2Direction := Tc2_MC2.MC_Direction.MC_Undefined_Direction;
        Tco_TO_Tc2MC2_Direction := TRUE;
ELSE
    Tco_TO_Tc2MC2_Direction := FALSE;
END_CASE

END_FUNCTION

// ---- POUs/Conversions/Tc2MC2_TO_Tco_Direction.TcPOU
FUNCTION INTERNAL Tc2MC2_TO_Tco_Direction : BOOL
VAR_INPUT
    Tc2MC2Direction : Tc2_MC2.MC_Direction;
END_VAR
VAR_IN_OUT
    TcoDirection : eDirection;
END_VAR

CASE Tc2MC2Direction OF
    Tc2_MC2.MC_Direction.MC_Current_Direction:
        TcoDirection := eDirection.MC_Current_Direction;
        Tc2MC2_TO_Tco_Direction := TRUE;
    Tc2_MC2.MC_Direction.MC_Negative_Direction:
        TcoDirection := eDirection.MC_Negative_Direction;
        Tc2MC2_TO_Tco_Direction := TRUE;
    Tc2_MC2.MC_Direction.MC_Positive_Direction:
        TcoDirection := eDirection.MC_Positive_Direction;
        Tc2MC2_TO_Tco_Direction := TRUE;
    Tc2_MC2.MC_Direction.MC_Shortest_Way:
        TcoDirection := eDirection.MC_Shortest_Way;
        Tc2MC2_TO_Tco_Direction := TRUE;
    Tc2_MC2.MC_Direction.MC_Undefined_Direction:
        TcoDirection := eDirection.MC_Undefined_Direction;
        Tc2MC2_TO_Tco_Direction := TRUE;
ELSE
    Tc2MC2_TO_Tco_Direction := FALSE;
END_CASE

END_FUNCTION

// ---- POUs/Conversions/Tco_TO_Tc2MC2_HomingMode.TcPOU
FUNCTION INTERNAL Tco_TO_Tc2MC2_HomingMode : BOOL
VAR_INPUT
    TcoHomingMode : eHomingMode;
END_VAR
VAR_IN_OUT
    Tc2MC2HomingMode : Tc2_MC2.MC_HomingMode;
END_VAR

CASE TcoHomingMode OF
    eHomingMode.MC_DefaultHoming:
        Tc2MC2HomingMode := Tc2_MC2.MC_HomingMode.MC_DefaultHoming;
        Tco_TO_Tc2MC2_HomingMode := TRUE;
    eHomingMode.MC_Direct:
        Tc2MC2HomingMode := Tc2_MC2.MC_HomingMode.MC_Direct;
        Tco_TO_Tc2MC2_HomingMode := TRUE;
    eHomingMode.MC_ForceCalibration:
        Tc2MC2HomingMode := Tc2_MC2.MC_HomingMode.MC_ForceCalibration;
        Tco_TO_Tc2MC2_HomingMode := TRUE;
    eHomingMode.MC_ResetCalibration:
        Tc2MC2HomingMode := Tc2_MC2.MC_HomingMode.MC_ResetCalibration;
        Tco_TO_Tc2MC2_HomingMode := TRUE;
ELSE
    Tco_TO_Tc2MC2_HomingMode := FALSE;
END_CASE

END_FUNCTION

// ---- POUs/Conversions/Tco_TO_Tc2MC2_EncRefMode.TcPOU
FUNCTION INTERNAL Tco_TO_Tc2MC2_EncRefMode : BOOL
VAR_INPUT
    TcoEncRef : eEncoderReferenceMode;
END_VAR
VAR_IN_OUT
    Tc2MC2EncRef : Tc2_MC2.E_EncoderReferenceMode;
END_VAR

CASE TcoEncRef OF
    eEncoderReferenceMode.ENCODERREFERENCEMODE_DEFAULT:
        Tc2MC2EncRef := Tc2_MC2.E_EncoderReferenceMode.ENCODERREFERENCEMODE_DEFAULT;
        Tco_TO_Tc2MC2_EncRefMode := TRUE;
    eEncoderReferenceMode.ENCODERREFERENCEMODE_PLCCAM:
        Tc2MC2EncRef := Tc2_MC2.E_EncoderReferenceMode.ENCODERREFERENCEMODE_PLCCAM;
        Tco_TO_Tc2MC2_EncRefMode := TRUE;
    eEncoderReferenceMode.ENCODERREFERENCEMODE_HARDWARESYNC:
        Tc2MC2EncRef := Tc2_MC2.E_EncoderReferenceMode.ENCODERREFERENCEMODE_HARDWARESYNC;
        Tco_TO_Tc2MC2_EncRefMode := TRUE;
    eEncoderReferenceMode.ENCODERREFERENCEMODE_HARDWARELATCHPOS:
        Tc2MC2EncRef := Tc2_MC2.E_EncoderReferenceMode.ENCODERREFERENCEMODE_HARDWARELATCHPOS;
        Tco_TO_Tc2MC2_EncRefMode := TRUE;
    eEncoderReferenceMode.ENCODERREFERENCEMODE_HARDWARELATCHNEG:
        Tc2MC2EncRef := Tc2_MC2.E_EncoderReferenceMode.ENCODERREFERENCEMODE_HARDWARELATCHNEG;
        Tco_TO_Tc2MC2_EncRefMode := TRUE;
    eEncoderReferenceMode.ENCODERREFERENCEMODE_SOFTWARESYNC:
        Tc2MC2EncRef := Tc2_MC2.E_EncoderReferenceMode.ENCODERREFERENCEMODE_SOFTWARESYNC;
        Tco_TO_Tc2MC2_EncRefMode := TRUE;
    eEncoderReferenceMode.ENCODERREFERENCEMODE_SOFTDRIVELATCHPOS:
        Tc2MC2EncRef := Tc2_MC2.E_EncoderReferenceMode.ENCODERREFERENCEMODE_SOFTDRIVELATCHPOS;
        Tco_TO_Tc2MC2_EncRefMode := TRUE;
    eEncoderReferenceMode.ENCODERREFERENCEMODE_SOFTDRIVELATCHNEG:
        Tc2MC2EncRef := Tc2_MC2.E_EncoderReferenceMode.ENCODERREFERENCEMODE_SOFTDRIVELATCHNEG;
        Tco_TO_Tc2MC2_EncRefMode := TRUE;
ELSE
    Tco_TO_Tc2MC2_EncRefMode := FALSE;
END_CASE

END_FUNCTION

// ---- POUs/Conversions/Tc2MC2_TO_Tco_EncRefMode.TcPOU
FUNCTION INTERNAL Tc2MC2_TO_Tco_EncRefMode : BOOL
VAR_INPUT
    Tc2MC2EncRef : Tc2_MC2.E_EncoderReferenceMode;
END_VAR
VAR_IN_OUT
    TcoEncRef : eEncoderReferenceMode;
END_VAR

CASE TcoEncRef OF
    Tc2_MC2.E_EncoderReferenceMode.ENCODERREFERENCEMODE_DEFAULT:
        TcoEncRef := eEncoderReferenceMode.ENCODERREFERENCEMODE_DEFAULT;
        Tc2MC2_TO_Tco_EncRefMode := TRUE;
    Tc2_MC2.E_EncoderReferenceMode.ENCODERREFERENCEMODE_PLCCAM:
        TcoEncRef := eEncoderReferenceMode.ENCODERREFERENCEMODE_PLCCAM;
        Tc2MC2_TO_Tco_EncRefMode := TRUE;
    Tc2_MC2.E_EncoderReferenceMode.ENCODERREFERENCEMODE_HARDWARESYNC:
        TcoEncRef := eEncoderReferenceMode.ENCODERREFERENCEMODE_HARDWARESYNC;
        Tc2MC2_TO_Tco_EncRefMode := TRUE;
    Tc2_MC2.E_EncoderReferenceMode.ENCODERREFERENCEMODE_HARDWARELATCHPOS:
        TcoEncRef := eEncoderReferenceMode.ENCODERREFERENCEMODE_HARDWARELATCHPOS;
        Tc2MC2_TO_Tco_EncRefMode := TRUE;
    Tc2_MC2.E_EncoderReferenceMode.ENCODERREFERENCEMODE_HARDWARELATCHNEG:
        TcoEncRef := eEncoderReferenceMode.ENCODERREFERENCEMODE_HARDWARELATCHNEG;
        Tc2MC2_TO_Tco_EncRefMode := TRUE;
    Tc2_MC2.E_EncoderReferenceMode.ENCODERREFERENCEMODE_SOFTWARESYNC:
        TcoEncRef := eEncoderReferenceMode.ENCODERREFERENCEMODE_SOFTWARESYNC;
        Tc2MC2_TO_Tco_EncRefMode := TRUE;
    Tc2_MC2.E_EncoderReferenceMode.ENCODERREFERENCEMODE_SOFTDRIVELATCHPOS:
        TcoEncRef := eEncoderReferenceMode.ENCODERREFERENCEMODE_SOFTDRIVELATCHPOS;
        Tc2MC2_TO_Tco_EncRefMode := TRUE;
    Tc2_MC2.E_EncoderReferenceMode.ENCODERREFERENCEMODE_SOFTDRIVELATCHNEG:
        TcoEncRef := eEncoderReferenceMode.ENCODERREFERENCEMODE_SOFTDRIVELATCHNEG;
        Tc2MC2_TO_Tco_EncRefMode := TRUE;
ELSE
    Tc2MC2_TO_Tco_EncRefMode := FALSE;
END_CASE

END_FUNCTION

// ---- POUs/Conversions/Tc2MC2_TO_Tco_HomingMode.TcPOU
FUNCTION INTERNAL Tc2MC2_TO_Tco_HomingMode : BOOL
VAR_INPUT
    Tc2MC2HomingMode : Tc2_MC2.MC_HomingMode;
END_VAR
VAR_IN_OUT
    TcoHomingMode : eHomingMode;
END_VAR

CASE Tc2MC2HomingMode OF
    Tc2_MC2.MC_HomingMode.MC_DefaultHoming:
        TcoHomingMode := eHomingMode.MC_DefaultHoming;
        Tc2MC2_TO_Tco_HomingMode := TRUE;
    Tc2_MC2.MC_HomingMode.MC_Direct:
        TcoHomingMode := eHomingMode.MC_Direct;
        Tc2MC2_TO_Tco_HomingMode := TRUE;
    Tc2_MC2.MC_HomingMode.MC_ForceCalibration:
        TcoHomingMode := eHomingMode.MC_ForceCalibration;
        Tc2MC2_TO_Tco_HomingMode := TRUE;
    Tc2_MC2.MC_HomingMode.MC_ResetCalibration:
        TcoHomingMode := eHomingMode.MC_ResetCalibration;
        Tc2MC2_TO_Tco_HomingMode := TRUE;
ELSE
    Tc2MC2_TO_Tco_HomingMode := FALSE;
END_CASE

END_FUNCTION

// ---- POUs/Conversions/Tco_TO_Tc2MC2_AxisStates.TcPOU
FUNCTION INTERNAL Tco_TO_Tc2MC2_AxisStates : BOOL
VAR_INPUT
    TcoAxisStates : eAxisStates;
END_VAR
VAR_IN_OUT
    Tc2MC2AxisStates : Tc2_MC2.MC_AxisStates;
END_VAR

CASE TcoAxisStates OF
    eAxisStates.MC_AXISSTATE_CONTINOUSMOTION:
        Tc2MC2AxisStates := Tc2_MC2.MC_AxisStates.MC_AXISSTATE_CONTINOUSMOTION;
        Tco_TO_Tc2MC2_AxisStates := TRUE;
    eAxisStates.MC_AXISSTATE_DISABLED:
        Tc2MC2AxisStates := Tc2_MC2.MC_AxisStates.MC_AXISSTATE_DISABLED;
        Tco_TO_Tc2MC2_AxisStates := TRUE;
    eAxisStates.MC_AXISSTATE_DISCRETEMOTION:
        Tc2MC2AxisStates := Tc2_MC2.MC_AxisStates.MC_AXISSTATE_DISCRETEMOTION;
        Tco_TO_Tc2MC2_AxisStates := TRUE;
    eAxisStates.MC_AXISSTATE_ERRORSTOP:
        Tc2MC2AxisStates := Tc2_MC2.MC_AxisStates.MC_AXISSTATE_ERRORSTOP;
        Tco_TO_Tc2MC2_AxisStates := TRUE;
    eAxisStates.MC_AXISSTATE_HOMING:
        Tc2MC2AxisStates := Tc2_MC2.MC_AxisStates.MC_AXISSTATE_HOMING;
        Tco_TO_Tc2MC2_AxisStates := TRUE;
    eAxisStates.MC_AXISSTATE_STANDSTILL:
        Tc2MC2AxisStates := Tc2_MC2.MC_AxisStates.MC_AXISSTATE_STANDSTILL;
        Tco_TO_Tc2MC2_AxisStates := TRUE;
    eAxisStates.MC_AXISSTATE_STOPPING:
        Tc2MC2AxisStates := Tc2_MC2.MC_AxisStates.MC_AXISSTATE_STOPPING;
        Tco_TO_Tc2MC2_AxisStates := TRUE;
    eAxisStates.MC_AXISSTATE_SYNCHRONIZEDMOTION:
        Tc2MC2AxisStates := Tc2_MC2.MC_AxisStates.MC_AXISSTATE_SYNCHRONIZEDMOTION;
        Tco_TO_Tc2MC2_AxisStates := TRUE;
    eAxisStates.MC_AXISSTATE_UNDEFINED:
        Tc2MC2AxisStates := Tc2_MC2.MC_AxisStates.MC_AXISSTATE_UNDEFINED;
        Tco_TO_Tc2MC2_AxisStates := TRUE;
ELSE
    Tco_TO_Tc2MC2_AxisStates := FALSE;
END_CASE

END_FUNCTION

// ---- POUs/Conversions/Tco_TO_Tc2MC2_JogMode.TcPOU
FUNCTION INTERNAL Tco_TO_Tc2MC2_JogMode : BOOL
VAR_INPUT
    TcoJogMode : eJogMode;
END_VAR
VAR_IN_OUT
    Tc2MC2JogMode : Tc2_MC2.E_JogMode;
END_VAR

CASE TcoJogMode OF
    eJogMode.MC_JOGMODE_STANDARD_SLOW:
        Tc2MC2JogMode := Tc2_MC2.E_JogMode.MC_JOGMODE_STANDARD_SLOW;
        Tco_TO_Tc2MC2_JogMode := TRUE;
    eJogMode.MC_JOGMODE_STANDARD_FAST:
        Tc2MC2JogMode := Tc2_MC2.E_JogMode.MC_JOGMODE_STANDARD_FAST;
        Tco_TO_Tc2MC2_JogMode := TRUE;
    eJogMode.MC_JOGMODE_CONTINOUS:
        Tc2MC2JogMode := Tc2_MC2.E_JogMode.MC_JOGMODE_CONTINOUS;
        Tco_TO_Tc2MC2_JogMode := TRUE;
    eJogMode.MC_JOGMODE_INCHING:
        Tc2MC2JogMode := Tc2_MC2.E_JogMode.MC_JOGMODE_INCHING;
        Tco_TO_Tc2MC2_JogMode := TRUE;
    eJogMode.MC_JOGMODE_INCHING_MODULO:
        Tc2MC2JogMode := Tc2_MC2.E_JogMode.MC_JOGMODE_INCHING_MODULO;
        Tco_TO_Tc2MC2_JogMode := TRUE;
ELSE
    Tco_TO_Tc2MC2_JogMode := FALSE;
END_CASE

END_FUNCTION

// ---- POUs/MAIN.TcPOU
PROGRAM MAIN
VAR
END_VAR

END_PROGRAM

// ---- POUs/Prototypes/CartesianCoordinateSystem/MultiAxisSystem/TcoMultiAxis.TcPOU
FUNCTION_BLOCK TcoMultiAxis EXTENDS TcoCore.TcoComponent IMPLEMENTS ITcoMultiAxis
VAR_INPUT
    inEnableAxis1 : BOOL;
    inEnablePositiveAxis1 : BOOL;
    inEnableNegativeAxis1 : BOOL;
    inCalibrationCamAxis1 : BOOL;
    refAxis1 : REFERENCE TO TcoAxisRef;
    inEnableAxis2 : BOOL;
    inEnablePositiveAxis2 : BOOL;
    inEnableNegativeAxis2 : BOOL;
    inCalibrationCamAxis2 : BOOL;
    refAxis2 : REFERENCE TO TcoAxisRef;
    inEnableAxis3 : BOOL;
    inEnablePositiveAxis3 : BOOL;
    inEnableNegativeAxis3 : BOOL;
    inCalibrationCamAxis3 : BOOL;
    refAxis3 : REFERENCE TO TcoAxisRef;
    inEnableAxis4 : BOOL;
    inEnablePositiveAxis4 : BOOL;
    inEnableNegativeAxis4 : BOOL;
    inCalibrationCamAxis4 : BOOL;
    refAxis4 : REFERENCE TO TcoAxisRef;
END_VAR
VAR_IN_OUT
    inoPositions : TcoMultiAxisPositionsRootContainer;
END_VAR
VAR
    {attribute 'hide'}
    _axis1Ref : REFERENCE TO TcoAxisRef;
    {attribute addProperty Name "<#Axis 1#>"}
    _axis1 : TcoDriveSimple(THIS^);
    {attribute 'hide'}
    _axis2Ref : REFERENCE TO TcoAxisRef;
    {attribute addProperty Name "<#Axis 2#>"}
    _axis2 : TcoDriveSimple(THIS^);
    {attribute 'hide'}
    _axis3Ref : REFERENCE TO TcoAxisRef;
    {attribute addProperty Name "<#Axis 3#>"}
    _axis3 : TcoDriveSimple(THIS^);
    {attribute 'hide'}
    _axis4Ref : REFERENCE TO TcoAxisRef;
    {attribute addProperty Name "<#Axis 4#>"}
    _axis4 : TcoDriveSimple(THIS^);
    {attribute addProperty Name "<#Status#>"}
    {attribute clr [ReadOnly()]}
    _status : TcoMultiAxisStatus;
    {attribute addProperty Name "<#Config#>"}
    _config : TcoMultiAxisConfig;
    {attribute addProperty Name "<#Load positions Task#>"}
    _loadPositionTask : TcoAxisExchangeDataTask(THIS^);
    {attribute addProperty Name "<#Save positions Task#>"}
    _savePositionTask : TcoAxisExchangeDataTask(THIS^);
    {attribute addProperty Name "<#Positions#>"}
    {attribute clr [MemberByIdentity()]}
    _positions : TcoMultiAxisPositionsRootContainer(THIS^);
    {attribute addProperty Name "<#Move Absolute Task#>"}
    _moveAbsoluteTask : TcoCore.TcoTask(THIS^);
    {attribute addProperty Name "<#Reset Drives Task#>"}
    _resetDrivesTask : TcoCore.TcoTask(THIS^);
    {attribute addProperty Name "<#Soe Reset Drives Task#>"}
    _soeResetDrivesTask : TcoCore.TcoTask(THIS^);
    {attribute addProperty Name "<#Abort Task#>"}
    _abortTask : TcoCore.TcoTask(THIS^);
    {attribute addProperty Name "<#Restore Task#>"}
    _restoreTask : TcoCore.TcoTask(THIS^);
    _moveParams : TcoMultiAxisMoveParam;
    _hasError : BOOL;
    {attribute 'hide'}
    _infoTimer : TON;
    {attribute 'hide'}
    _errorTimer : TON;
    _done : BOOL;
    _override : LREAL;
END_VAR

_positions := inoPositions;
//****************************************
_savePositionTask();
_loadPositionTask();
_abortTask.Enabled := TRUE;

//*************Abort Task********************
IF _abortTask.Execute() THEN
    IF NOT _config.Axis1Disabled THEN
        THIS^._axis1.MoveAbosluteAbort();
    END_IF;

    IF NOT _config.Axis2Disabled THEN
        THIS^._axis2.MoveAbosluteAbort();
    END_IF;

    IF NOT _config.Axis3Disabled THEN
        THIS^._axis3.MoveAbosluteAbort();
    END_IF;

    IF NOT _config.Axis4Disabled THEN
        THIS^._axis4.MoveAbosluteAbort();
    END_IF;

    _abortTask.DoneWhen(TRUE);
    _abortTask.ThrowWhen(_hasError);
END_IF;
//****************************************
//*************RESTORE********************
_restoreTask.Enabled := TRUE;

IF _restoreTask.Execute() THEN
    Restore();
END_IF

//****************************************
IF NOT __ISVALIDREF(refAxis1) AND NOT _config.Axis1Disabled THEN
    Messenger.Post('<#Invalid reference axis 1#>', TcoCore.eMessageCategory.ProgrammingError);
    RETURN;
ELSIF NOT _config.Axis1Disabled THEN
    _axis1Ref REF= refAxis1;

    _axis1(inEnable := inEnableAxis1,
        inEnablePositive := inEnablePositiveAxis1,
        inEnableNegative := inEnableNegativeAxis1,
        inCalibrationCam := inCalibrationCamAxis1,
        inoAxisRef := _axis1Ref);
END_IF

IF NOT __ISVALIDREF(refAxis2) AND NOT _config.Axis2Disabled THEN
    Messenger.Post('<#Invalid reference axis 2#>', TcoCore.eMessageCategory.ProgrammingError);
    RETURN;
ELSIF NOT _config.Axis2Disabled THEN
    _axis2Ref REF= refAxis2;

    _axis2(inEnable := inEnableAxis2,
        inEnablePositive := inEnablePositiveAxis2,
        inEnableNegative := inEnableNegativeAxis2,
        inCalibrationCam := inCalibrationCamAxis2,
        inoAxisRef := _axis2Ref);
END_IF

IF NOT __ISVALIDREF(refAxis3) AND NOT _config.Axis3Disabled THEN
    Messenger.Post('<#Invalid reference axis 3#>', TcoCore.eMessageCategory.ProgrammingError);
    RETURN;
ELSIF NOT _config.Axis3Disabled THEN
    _axis3Ref REF= refAxis3;

    _axis3(inEnable := inEnableAxis3,
        inEnablePositive := inEnablePositiveAxis3,
        inEnableNegative := inEnableNegativeAxis3,
        inCalibrationCam := inCalibrationCamAxis3,
        inoAxisRef := _axis3Ref);
END_IF

IF NOT __ISVALIDREF(refAxis4) AND NOT _config.Axis4Disabled THEN
    Messenger.Post('<#Invalid reference axis 4#>', TcoCore.eMessageCategory.ProgrammingError);
    RETURN;
ELSIF NOT _config.Axis4Disabled THEN
    _axis4Ref REF= refAxis4;

    _axis4(inEnable := inEnableAxis4,
        inEnablePositive := inEnablePositiveAxis4,
        inEnableNegative := inEnableNegativeAxis4,
        inCalibrationCam := inCalibrationCamAxis4,
        inoAxisRef := _axis4Ref);
END_IF
//*************MOVE ABSOLUTE********************
_moveAbsoluteTask.Enabled := NOT _resetDrivesTask.Busy AND NOT _soeResetDrivesTask.Busy;

IF _moveAbsoluteTask.Execute() THEN
    IF NOT _config.Axis1Disabled THEN
        THIS^._axis1.MoveAbsolute(inPosition := _moveParams.Axis1.Position,
            inVelocity := _moveParams.Axis1.Velocity,
            inAcceleration := _moveParams.Axis1.Acceleration,
            inDeceleration := _moveParams.Axis1.Deceleration,
            inJerk := _moveParams.Axis1.Jerk);
    END_IF;

    IF NOT _config.Axis2Disabled THEN
        THIS^._axis2.MoveAbsolute(inPosition := _moveParams.Axis2.Position,
            inVelocity := _moveParams.Axis2.Velocity,
            inAcceleration := _moveParams.Axis2.Acceleration,
            inDeceleration := _moveParams.Axis2.Deceleration,
            inJerk := _moveParams.Axis2.Jerk);
    END_IF;

    IF NOT _config.Axis3Disabled THEN
        THIS^._axis3.MoveAbsolute(inPosition := _moveParams.Axis3.Position,
            inVelocity := _moveParams.Axis3.Velocity,
            inAcceleration := _moveParams.Axis3.Acceleration,
            inDeceleration := _moveParams.Axis3.Deceleration,
            inJerk := _moveParams.Axis3.Jerk);
    END_IF;

    IF NOT _config.Axis4Disabled THEN
        THIS^._axis4.MoveAbsolute(inPosition := _moveParams.Axis4.Position,
            inVelocity := _moveParams.Axis4.Velocity,
            inAcceleration := _moveParams.Axis4.Acceleration,
            inDeceleration := _moveParams.Axis4.Deceleration,
            inJerk := _moveParams.Axis4.Jerk);
    END_IF;

    _hasError := (THIS^._axis1.MoveAbsoluteTask.Error AND NOT _config.Axis1Disabled) OR
        (THIS^._axis2.MoveAbsoluteTask.Error AND NOT _config.Axis2Disabled) OR
        (THIS^._axis3.MoveAbsoluteTask.Error AND NOT _config.Axis3Disabled) OR
        (THIS^._axis4.MoveAbsoluteTask.Error AND NOT _config.Axis4Disabled);

    _done := (THIS^._axis1.MoveAbsoluteTask.Done OR _config.Axis1Disabled) AND
        (THIS^._axis2.MoveAbsoluteTask.Done OR _config.Axis2Disabled) AND
        (THIS^._axis3.MoveAbsoluteTask.Done OR _config.Axis3Disabled) AND
        (THIS^._axis4.MoveAbsoluteTask.Done OR _config.Axis4Disabled);

    _moveAbsoluteTask.DoneWhen(_done);
    _moveAbsoluteTask.ThrowWhen(_hasError);
END_IF;
//*************Reset Drives********************
_resetDrivesTask.Enabled := NOT _moveAbsoluteTask.Busy AND NOT _soeResetDrivesTask.Busy;

IF _resetDrivesTask.Execute() THEN
    IF NOT _config.Axis1Disabled THEN
        THIS^._axis1.Reset();
    END_IF;

    IF NOT _config.Axis2Disabled THEN
        THIS^._axis2.Reset();
    END_IF;

    IF NOT _config.Axis3Disabled THEN
        THIS^._axis3.Reset();
    END_IF;

    IF NOT _config.Axis4Disabled THEN
        THIS^._axis4.Reset();
    END_IF;

    _hasError := (THIS^._axis1.ResetTask.Error AND NOT _config.Axis1Disabled) OR
        (THIS^._axis2.ResetTask.Error AND NOT _config.Axis2Disabled) OR
        (THIS^._axis3.ResetTask.Error AND NOT _config.Axis3Disabled) OR
        (THIS^._axis4.ResetTask.Error AND NOT _config.Axis4Disabled);

    _done := (THIS^._axis1.ResetTask.Done XOR _config.Axis1Disabled) AND
        (THIS^._axis2.ResetTask.Done XOR _config.Axis2Disabled) AND
        (THIS^._axis3.ResetTask.Done XOR _config.Axis3Disabled) AND
        (THIS^._axis4.ResetTask.Done XOR _config.Axis4Disabled);

    _resetDrivesTask.DoneWhen(_done);
    _resetDrivesTask.ThrowWhen(_hasError);
END_IF;

_soeResetDrivesTask.Enabled := NOT _moveAbsoluteTask.Busy AND NOT _ResetDrivesTask.Busy;

//*************Soe Reset Drives********************
IF _soeResetDrivesTask.Execute() THEN
    IF NOT _config.Axis1Disabled THEN
        THIS^._axis1.SoEReset();
    END_IF;

    IF NOT _config.Axis2Disabled THEN
        THIS^._axis2.SoeReset();
    END_IF;

    IF NOT _config.Axis3Disabled THEN
        THIS^._axis3.SoEReset();
    END_IF;

    IF NOT _config.Axis4Disabled THEN
        THIS^._axis4.SoEReset();
    END_IF;

    _hasError := (THIS^._axis1.SoEResetTask.Error AND NOT _config.Axis1Disabled) OR
        (THIS^._axis2.SoEResetTask.Error AND NOT _config.Axis2Disabled) OR
        (THIS^._axis3.SoEResetTask.Error AND NOT _config.Axis3Disabled) OR
        (THIS^._axis4.SoEResetTask.Error AND NOT _config.Axis4Disabled);

    _done := (THIS^._axis1.SoEResetTask.Done XOR _config.Axis1Disabled) AND
        (THIS^._axis2.SoEResetTask.Done XOR _config.Axis2Disabled) AND
        (THIS^._axis3.SoEResetTask.Done XOR _config.Axis3Disabled) AND
        (THIS^._axis4.ResetTask.Done XOR _config.Axis4Disabled);

    _soeResetDrivesTask.DoneWhen(_done);
    _soeResetDrivesTask.ThrowWhen(_errorTimer.Q OR _hasError);
END_IF;

inoPositions := _positions;

PROPERTY PUBLIC AbortTask : REFERENCE TO TcoCore.TcoTask
GET
AbortTask REF= _abortTask;
END_GET
END_PROPERTY

PROPERTY Axis_1 : REFERENCE TO TcoDriveSimple
GET
Axis_1 REF= _axis1;
END_GET
END_PROPERTY

PROPERTY Axis_2 : REFERENCE TO TcoDriveSimple
GET
Axis_2 REF= _axis2;
END_GET
END_PROPERTY

PROPERTY Axis_3 : REFERENCE TO TcoDriveSimple
GET
Axis_3 REF= _axis3;
END_GET
END_PROPERTY

PROPERTY Axis_4 : REFERENCE TO TcoDriveSimple
GET
Axis_4 REF= _axis4;
END_GET
END_PROPERTY

METHOD CallTimers
VAR_INPUT
    inValue : BOOL;
END_VAR
IF __ISVALIDREF(Config) THEN
    _infoTimer(IN := inValue, PT := THIS^.Config.InfoTime);
    _errorTimer(IN := inValue, PT := THIS^.Config.ErrorTime);
END_IF;
END_METHOD

(*~
    <docu>
        <summary>
            Gets the configuration of the SFK.
        </summary>
    </docu>
~*)
PROPERTY Config : REFERENCE TO TcoMultiAxisConfig
GET
Config REF= _config;
END_GET
END_PROPERTY

PROPERTY PUBLIC LoadPositionsTask : REFERENCE TO TcoAxisExchangeDataTask
GET
LoadPositionsTask REF= _loadPositionTask;
END_GET
END_PROPERTY

METHOD MoveAbsolute : TcoCore.ITcoTaskStatus
VAR_INPUT
    MoveParams : TcoMultiAxisMoveParam;
END_VAR
_moveParams := MoveParams;
MoveAbsolute := THIS^._moveAbsoluteTask.Invoke();
END_METHOD

PROPERTY PUBLIC MoveAbsoluteTask : REFERENCE TO TcoCore.TcoTask
GET
MoveAbsoluteTask REF= _moveAbsoluteTask;
END_GET
END_PROPERTY

METHOD ResetDrives : TcoCore.ITcoTaskStatus
ResetDrives := THIS^._resetDrivesTask.Invoke();
END_METHOD

PROPERTY PUBLIC ResetDrivesTask : REFERENCE TO TcoCore.TcoTask
GET
ResetDrivesTask REF= _resetDrivesTask;
END_GET
END_PROPERTY

(*~
    <docu>
        <summary>
            Restores this instance to the Ready state. Can be called explicitly or from within one of the restore mechanisms.
        </summary>
    </docu>
~*)
METHOD Restore : ITcoRestorable
_axis1.Restore();
_axis2.Restore();
_axis3.Restore();
_axis4.Restore();
_restoreTask.Restore();
_abortTask.Restore();
_savePositionTask.Restore();
_loadPositionTask.Restore();
_moveAbsoluteTask.Restore();
_soeResetDrivesTask.Restore();
_resetDrivesTask.Restore();
CallTimers(FALSE);
Messenger.UnPin();
END_METHOD

PROPERTY PUBLIC SavePositionsTask : REFERENCE TO TcoAxisExchangeDataTask
GET
SavePositionsTask REF= _savePositionTask;
END_GET
END_PROPERTY

METHOD PROTECTED ServiceMode
THIS^._axis1.Service();
THIS^._axis2.Service();
THIS^._axis3.Service();
THIS^._axis4.Service();
END_METHOD

METHOD SoeReset : TcoCore.ITcoTaskStatus
SoeReset := THIS^._soeResetDrivesTask.Invoke();
END_METHOD

PROPERTY PUBLIC SoeResetDrivesTask : REFERENCE TO TcoCore.TcoTask
GET
SoeResetDrivesTask REF= _soeResetDrivesTask;
END_GET
END_PROPERTY

(*~
    <docu>
        <summary>
            Gets the status of the TcoMultiAxis system.
        </summary>
    </docu>
~*)
PROPERTY Status : REFERENCE TO TcoMultiAxisStatus
GET
Status REF= _status;
END_GET
END_PROPERTY

END_FUNCTION_BLOCK

// ---- POUs/Prototypes/CartesianCoordinateSystem/MultiAxisSystem/TcoMultiAxisPositionsRootContainer.TcPOU
FUNCTION_BLOCK TcoMultiAxisPositionsRootContainer EXTENDS TcoCore.TcoObject
VAR_INPUT
END_VAR
VAR_OUTPUT
END_VAR
VAR
END_VAR

END_FUNCTION_BLOCK

// ---- POUs/Prototypes/TcoDriveSimple/TcoDriveSimple.TcPOU
FUNCTION_BLOCK TcoDriveSimple EXTENDS TcoCore.TcoComponent IMPLEMENTS ITcoDriveSimple
VAR_INPUT
    inEnable : BOOL;
    inEnablePositive : BOOL;
    inEnableNegative : BOOL;
    inCalibrationCam : BOOL;
END_VAR
VAR_OUTPUT
END_VAR
VAR_IN_OUT
    inoAxisRef : TcoAxisRef;
END_VAR
VAR
    {attribute 'hide'}
    _axisRef : REFERENCE TO TcoAxisRef;
    {attribute 'hide'}
    _mcReadStatus : Tc2_MC2.MC_ReadStatus;
    _override : LREAL := 100.0;
    {attribute 'hide'}
    _overrideInternal : LREAL := 100.0;
    {attribute addProperty Name "<#Axis status#>"}
    {attribute clr [ReadOnly()]}
    _axisStatus : TcoAxisStatus;
    {attribute addProperty Name "<#Axis config#>"}
    _config : TcoAxisConfig;
    _reduceMovementsInServiceMode : REAL;
END_VAR
VAR
    {attribute addProperty Name "<#Movement state#>"}
    {attribute clr [ReadOnly()]}
    _movementState : TcoMovementState(THIS^, TcoCore.eRestoreMode.None);
    {attribute addProperty Name "<#Power#>"}
    _power : Power(THIS^);
    {attribute addProperty Name "<#Reset#>"}
    _resetTask : ResetTask(THIS^);
    {attribute addProperty Name "<#SoE reset#>"}
    _soEResetTask : SoEResetTask(THIS^);
    {attribute addProperty Name "<#Set position#>"}
    _setPositionTask : SetPositionTask(THIS^);
    {attribute addProperty Name "<#Homing#>"}
    _homeTask : HomeTask(THIS^);
    {attribute addProperty Name "<#Jogging#>"}
    _jog : Jog(THIS^);
    {attribute addProperty Name "<#Force/Torque#>"}
    _torqueTask : SetTorqueTask(THIS^);
    {attribute addProperty Name "<#Move velocity#>"}
    _moveVelocityTask : MoveVelocityTask(THIS^);
    {attribute addProperty Name "<#Stop#>"}
    _stopTask : StopTask(THIS^);
    {attribute addProperty Name "<#Halt#>"}
    _haltTask : HaltTask(THIS^);
    {attribute addProperty Name "<#Move relative#>"}
    _moveRelativeTask : MoveRelativeTask(THIS^);
    {attribute addProperty Name "<#Move absolute#>"}
    _moveAbsoluteTask : MoveAbsoluteTask(THIS^);
    {attribute addProperty Name "<#Move modulo#>"}
    _moveModuloTask : MoveModuloTask(THIS^);
END_VAR
VAR
    {attribute 'hide'}
    _sb : TcoCore.StringBuilder;
END_VAR

IF NOT __ISVALIDREF(inoAxisRef) THEN
    Messenger.Post('Invalid reference', TcoCore.eMessageCategory.ProgrammingError);
    RETURN;
END_IF

_axisRef REF= inoAxisRef;
_mcReadStatus(Axis := _axisRef, Enable := TRUE);
UpdateAxisStatus();
_overrideInternal := _override;

IF _config.OverrideInService > 0.0 AND _config.OverrideInService <= 100.0 AND THIS^.IsService THEN
    _overrideInternal := _config.OverrideInService;

    Messenger.Notify(_sb.Clear()
            .Append('<#Drive in override mode (Reduced velocity) due service mode! Limited to #>')
            .Append(LREAL_TO_STRING(_overrideInternal))
            .Append(' %')
            .ToString());
END_IF

_power(inEnable := inEnable,
    inEnablePositive := inEnablePositive,
    inEnableNegative := inEnableNegative,
    inOverride := _overrideInternal,
    inIsServiceMode := THIS^.IsService);

_resetTask();
_soEResetTask();
_setPositionTask();
_homeTask();
_jog(inIsServiceMode := THIS^.IsService);
_moveVelocityTask();
_stopTask();
_haltTask();
_moveRelativeTask();
_moveAbsoluteTask();
_moveModuloTask();
_torqueTask(inIsServiceMode := THIS^.IsService);

IF (_axisStatus.Error) THEN
    Messenger.Error(_sb.Clear()
            .Append('<#Drive error no #>')
            .Append(UDINT_TO_STRING(_axisStatus.ErrorId))
            .Append(' |[[0]AdvancedDiagnosticMessage]|')
            .Append('.')
            .Append('For details see the service mode')
            .ToString());
END_IF;

PROPERTY AxisRef : REFERENCE TO TcoAxisRef
GET
IF __ISVALIDREF(_axisRef) THEN
    AxisRef REF= _axisRef;
END_IF;
END_GET
END_PROPERTY

PROPERTY AxisStatus : REFERENCE TO TcoAxisStatus
GET
UpdateAxisStatus();
AxisStatus REF= _axisStatus;
END_GET
END_PROPERTY

METHOD INTERNAL ClearError
_axisStatus.Error := FALSE;
_axisStatus.ErrorId := 0;
END_METHOD

(*~
    <docu>
        <summary>
            Gets the configuration of the Axis.
        </summary>
    </docu>
~*)
PROPERTY Config : REFERENCE TO TcoAxisConfig
GET
Config REF= _config;
END_GET
END_PROPERTY

PROPERTY DriveRef : REFERENCE TO TcoDriveSimple
GET
DriveRef REF= THIS^;
END_GET
END_PROPERTY

METHOD FB_init : BOOL
VAR_INPUT
    bInitRetains : BOOL; // if TRUE, the retain variables are initialized (warm start / cold start)
    bInCopyCode : BOOL; // if TRUE, the instance afterwards gets moved into the copy code (online change)
    ParentObject : ITcoObject;
END_VAR
END_METHOD

METHOD Halt : ITcoTaskStatus
VAR_INPUT
    inDeceleration : LREAL;
    inJerk : LREAL;
END_VAR
Halt := THIS^._haltTask.InvokeWithParams(inDeceleration := inDeceleration, inJerk := inJerk);
END_METHOD

PROPERTY HaltTask : TcoCore.ITcoTaskStatus
GET
HaltTask := _haltTask;
END_GET
END_PROPERTY

METHOD Home : ITcoTaskStatus
VAR_INPUT
    inPosition : LREAL;
    inHomingMode : eHomingMode;
    inClearPositionLag : BOOL;
    inSearchDirection : eDirection;
    inSearchVelocity : LREAL;
    inSyncDirection : eDirection;
    inSyncVelocity : LREAL;
    inReferenceMode : eEncoderReferenceMode;
END_VAR
Home := THIS^._homeTask.InvokeWithParams(inPosition := inPosition,
    inHomingMode := inHomingMode,
    inClearPositionLag := inClearPositionLag,
    inSearchDirection := inSearchDirection,
    inSearchVelocity := inSearchVelocity,
    inSyncDirection := inSyncDirection,
    inSyncVelocity := inSyncVelocity,
    inReferenceMode := inReferenceMode);
END_METHOD

METHOD PUBLIC HomeAbort
VAR_INPUT
END_VAR
_homeTask.Abort();
END_METHOD

PROPERTY HomeTask : TcoCore.ITcoTaskStatus
GET
HomeTask := _homeTask;
END_GET
END_PROPERTY

METHOD PUBLIC InPosition : BOOL
VAR_INPUT
    inRequiredPos : LREAL;
    inWindow : LREAL;
END_VAR
InPosition := ABS(_axisStatus.ActPos - inRequiredPos) < inWindow;
END_METHOD

PROPERTY IsEnabled : BOOL
GET
IsEnabled := inEnable AND _axisStatus.Operational;
END_GET
END_PROPERTY

PROPERTY IsEnabledNegative : BOOL
GET
IsEnabledNegative := inEnableNegative;
END_GET
END_PROPERTY

PROPERTY IsEnabledPositive : BOOL
GET
IsEnabledPositive := inEnablePositive;
END_GET
END_PROPERTY

METHOD PUBLIC MoveAbosluteAbort
VAR_INPUT
END_VAR
_moveAbsoluteTask.Abort();
END_METHOD

METHOD MoveAbsolute : ITcoTaskStatus
VAR_INPUT
    inPosition : LREAL;
    inVelocity : LREAL;
    inAcceleration : LREAL;
    inDeceleration : LREAL;
    inJerk : LREAL;
END_VAR
MoveAbsolute := THIS^._moveAbsoluteTask.InvokeWithParams(inPosition := inPosition,
    inVelocity := inVelocity,
    inAcceleration := inAcceleration,
    inDeceleration := inDeceleration,
    inJerk := inJerk);
END_METHOD

PROPERTY MoveAbsoluteTask : TcoCore.ITcoTaskStatus
GET
MoveAbsoluteTask := _moveAbsoluteTask;
END_GET
END_PROPERTY

METHOD MoveModulo : ITcoTaskStatus
VAR_INPUT
    inPosition : LREAL;
    inVelocity : LREAL;
    inAcceleration : LREAL;
    inDeceleration : LREAL;
    inJerk : LREAL;
    inDirection : eDirection;
END_VAR
MoveModulo := THIS^._moveModuloTask.InvokeWithParams(inPosition := inPosition,
    inVelocity := inVelocity,
    inAcceleration := inAcceleration,
    inDeceleration := inDeceleration,
    inJerk := inJerk,
    inDirection := inDirection);
END_METHOD

PROPERTY MoveModuloTask : TcoCore.ITcoTaskStatus
GET
MoveModuloTask := _moveModuloTask;
END_GET
END_PROPERTY

METHOD MoveRelative : ITcoTaskStatus
VAR_INPUT
    inDistance : LREAL;
    inVelocity : LREAL;
    inAcceleration : LREAL;
    inDeceleration : LREAL;
    inJerk : LREAL;
END_VAR
MoveRelative := THIS^._moveRelativeTask.InvokeWithParams(inDistance := inDistance,
    inVelocity := inVelocity,
    inAcceleration := inAcceleration,
    inDeceleration := inDeceleration,
    inJerk := inJerk);
END_METHOD

PROPERTY MoveRelativeTask : TcoCore.ITcoTaskStatus
GET
MoveRelativeTask := _moveRelativeTask;
END_GET
END_PROPERTY

METHOD MoveVelocity : ITcoTaskStatus
VAR_INPUT
    inVelocity : LREAL;
    inAcceleration : LREAL;
    inDeceleration : LREAL;
    inJerk : LREAL;
    inDirection : eDirection;
END_VAR
MoveVelocity := THIS^._moveVelocityTask.InvokeWithParams(inVelocity := inVelocity,
    inAcceleration := inAcceleration,
    inDeceleration := inDeceleration,
    inJerk := inJerk,
    inDirection := inDirection);
END_METHOD

PROPERTY MoveVelocityTask : TcoCore.ITcoTaskStatus
GET
MoveVelocityTask := _moveVelocityTask;
END_GET
END_PROPERTY

(*~
        <docu>
            <summary>
            Velocity override in % FOR all movement commands. (0 ≤ Override ≤ 100.0)
            </summary>
        </docu>
~*)
PROPERTY Override : LREAL
GET
Override := _override;
END_GET
SET
_override := Override;
END_SET
END_PROPERTY

METHOD Reset : ITcoTaskStatus
Reset := THIS^._resetTask.Invoke();
END_METHOD

PROPERTY ResetTask : TcoCore.ITcoTaskStatus
GET
ResetTask := _resetTask;
END_GET
END_PROPERTY

(*~
    <docu>
        <summary>
            Restores this instance to the Ready state. Can be called explicitly or from within one of the restore mechanisms.
        </summary>
    </docu>
~*)
METHOD Restore : ITcoRestorable
IF __ISVALIDREF(_axisRef) THEN
    IF NOT inEnable THEN
        _Power(inEnable := FALSE);
    END_IF

    _mcReadStatus(Axis := _axisRef, Enable := FALSE);
END_IF

IF NOT (_override > 0.0 AND _override <= 100.0) THEN
    _override := 100;
END_IF

RestoreTasks();
_resetTask.Restore();
END_METHOD

METHOD INTERNAL RestoreTasks
//_resetTask.Restore();
_soEResetTask.Restore();
_setPositionTask.Restore();
_homeTask.Restore();
_moveVelocityTask.Restore();
_stopTask.Restore();
_haltTask.Restore();
_moveRelativeTask.Restore();
_moveAbsoluteTask.Restore();
_moveModuloTask.Restore();
_movementState.Restore();
_torqueTask.Restore();
END_METHOD

(*~
    <docu>
        <summary>
            Custom service (manual, maintenance) logic.
            This method must be implemented in derived class.
        </summary>
    </docu>
~*)
METHOD PROTECTED ServiceMode
_jog.Service();
END_METHOD

METHOD INTERNAL SetErrorID
VAR_INPUT
    inErrorId : UDINT;
END_VAR
_axisStatus.Error := TRUE;

IF inErrorId <> 0 THEN
    _axisStatus.ErrorId := inErrorId;
END_IF
END_METHOD

METHOD SetPosition : ITcoTaskStatus
VAR_INPUT
    inPosition : LREAL;
    inMode : eSetPositionMode;
END_VAR
SetPosition := THIS^._setPositionTask.InvokeWithParams(inPosition := inPosition, inMode := inMode);
END_METHOD

PROPERTY SetPositionTask : TcoCore.ITcoTaskStatus
GET
SetPositionTask := _setPositionTask;
END_GET
END_PROPERTY

METHOD SetTorque : ITcoTaskStatus
VAR_INPUT
    inTorque : LREAL;
    inRelative : BOOL;
    inVelocityLimitHigh : LREAL;
    inVelocityLimitLow : LREAL;
    inContinuousUpdate : BOOL := TRUE;
    inTorqueRamp : LREAL;
    inTorqueOptions : Tc2_MC2.ST_TorqueControlOptions;
END_VAR
SetTorque := THIS^._torqueTask.InvokeWithParams(inTorque := inTorque,
    inRelative := inRelative,
    inVelocityLimitHigh := inVelocityLimitHigh,
    inVelocityLimitLow := inVelocityLimitLow,
    inContinuousUpdate := inContinuousUpdate,
    inTorqueRamp := inTorqueRamp,
    inTorqueOptions := inTorqueOptions);
END_METHOD

PROPERTY SetTorqueTask : TcoCore.ITcoTaskStatus
GET
SetTorqueTask := _torqueTask;
END_GET
END_PROPERTY

METHOD SoEReset : ITcoTaskStatus
SoEReset := THIS^._soEResetTask.Invoke();
END_METHOD

PROPERTY SoEResetTask : TcoCore.ITcoTaskStatus
GET
SoEResetTask := _soEResetTask;
END_GET
END_PROPERTY

METHOD Stop : ITcoTaskStatus
VAR_INPUT
    inDeceleration : LREAL;
    inJerk : LREAL;
END_VAR
Stop := THIS^._stopTask.InvokeWithParams(inDeceleration := inDeceleration, inJerk := inJerk);
END_METHOD

PROPERTY StopTask : TcoCore.ITcoTaskStatus
GET
StopTask := _stopTask;
END_GET
END_PROPERTY

METHOD INTERNAL UpdateAxisStatus
VAR
    _message : STRING(125);
END_VAR
_axisStatus.ActPos := AxisRef.NcToPlc.ActPos;
_axisStatus.ModuloActPos := AxisRef.NcToPlc.ModuloActPos;
_axisStatus.ModuloActTurns := AxisRef.NcToPlc.ModuloActTurns;
_axisStatus.ActVelo := AxisRef.NcToPlc.ActVelo;
_axisStatus.ActAcc := AxisRef.NcToPlc.ActAcc;
_axisStatus.ActTorque := AxisRef.NcToPlc.ActTorque;
_axisStatus.CmdNo := AxisRef.NcToPlc.CmdNo;
_axisStatus.CmdState := AxisRef.NcToPlc.CmdState;

IF NOT Tc2MC2_TO_Tco_AxisStates(AxisRef.Status.MotionState, _axisStatus.MotionState) THEN
    _message := Tc2_Standard
        .CONCAT('Unable to cast AxisRef.Status.MotionState variable of type Tc2_MC2.MC_AxisStates (', TO_STRING(AxisRef.Status.MotionState));

    _message := Tc2_Standard.CONCAT(_message, ') to the type TcoDrivesBeckhoff.eAxisStates!!!');
    THIS^.Messenger.Post(_message, TcoCore.eMessageCategory.ProgrammingError);
END_IF

IF AxisRef.Status.Error THEN
    _axisStatus.Error := AxisRef.Status.Error;
    _axisStatus.ErrorId := AxisRef.Status.ErrorId;
END_IF;

_axisStatus.ErrorStop := AxisRef.Status.ErrorStop;
_axisStatus.Disabled := AxisRef.Status.Disabled;
_axisStatus.Stopping := AxisRef.Status.Stopping;
_axisStatus.StandStill := AxisRef.Status.StandStill;
_axisStatus.DiscreteMotion := AxisRef.Status.DiscreteMotion;
_axisStatus.ContinuousMotion := AxisRef.Status.ContinuousMotion;
_axisStatus.SynchronizedMotion := AxisRef.Status.SynchronizedMotion;
_axisStatus.Homing := AxisRef.Status.Homing;
_axisStatus.ConstantVelocity := AxisRef.Status.ConstantVelocity;
_axisStatus.Accelerating := AxisRef.Status.Accelerating;
_axisStatus.Decelerating := AxisRef.Status.Decelerating;
_axisStatus.Operational := AxisRef.Status.Operational;
_axisStatus.ControlLoopClosed := AxisRef.Status.ControlLoopClosed;
_axisStatus.HasJob := AxisRef.Status.HasJob;
_axisStatus.HasBeenStopped := AxisRef.Status.HasBeenStopped;
_axisStatus.NewTargetPosition := AxisRef.Status.NewTargetPosition;
_axisStatus.InPositionArea := AxisRef.Status.InPositionArea;
_axisStatus.InTargetPosition := AxisRef.Status.InTargetPosition;
_axisStatus.Homed := AxisRef.Status.Homed;
_axisStatus.HomingBusy := AxisRef.Status.HomingBusy;
_axisStatus.MotionCommandsLocked := AxisRef.Status.MotionCommandsLocked;
_axisStatus.SoftLimitMinExceeded := AxisRef.Status.SoftLimitMinExceeded;
_axisStatus.SoftLimitMaxExceeded := AxisRef.Status.SoftLimitMaxExceeded;
_axisStatus.Moving := AxisRef.Status.Moving;
_axisStatus.PositiveDirection := AxisRef.Status.PositiveDirection;
_axisStatus.NegativeDirection := AxisRef.Status.NegativeDirection;
_axisStatus.NotMoving := AxisRef.Status.NotMoving;
_axisStatus.Compensating := AxisRef.Status.Compensating;
_axisStatus.ExtSetPointGenEnabled := AxisRef.Status.ExtSetPointGenEnabled;
_axisStatus.ExternalLatchValid := AxisRef.Status.ExternalLatchValid;
_axisStatus.CamDataQueued := AxisRef.Status.CamDataQueued;
_axisStatus.CamTableQueued := AxisRef.Status.CamTableQueued;
_axisStatus.CamScalingPending := AxisRef.Status.CamScalingPending;
_axisStatus.CmdBuffered := AxisRef.Status.CmdBuffered;
_axisStatus.PTPmode := AxisRef.Status.PTPmode;
_axisStatus.DriveDeviceError := AxisRef.Status.DriveDeviceError;
_axisStatus.IoDataInvalid := AxisRef.Status.IoDataInvalid;
_axisStatus.Coupled := AxisRef.Status.Coupled;
_axisStatus.OpMode.PositionAreaMonitoring := AxisRef.Status.OpMode.PositionAreaMonitoring;
_axisStatus.OpMode.TargetPositionMonitoring := AxisRef.Status.OpMode.TargetPositionMonitoring;
_axisStatus.OpMode.LoopMode := AxisRef.Status.OpMode.LoopMode;
_axisStatus.OpMode.MotionMonitoring := AxisRef.Status.OpMode.MotionMonitoring;
_axisStatus.OpMode.PEHTimeMonitoring := AxisRef.Status.OpMode.PEHTimeMonitoring;
_axisStatus.OpMode.BacklashCompensation := AxisRef.Status.OpMode.BacklashCompensation;
_axisStatus.OpMode.Modulo := AxisRef.Status.OpMode.Modulo;
_axisStatus.OpMode.PositionLagMonitoring := AxisRef.Status.OpMode.PositionLagMonitoring;
_axisStatus.OpMode.VelocityLagMonitoring := AxisRef.Status.OpMode.VelocityLagMonitoring;
_axisStatus.OpMode.SoftLimitMinMonitoring := AxisRef.Status.OpMode.SoftLimitMinMonitoring;
_axisStatus.OpMode.SoftLimitMaxMonitoring := AxisRef.Status.OpMode.SoftLimitMaxMonitoring;
_axisStatus.OpMode.PositionCorrection := AxisRef.Status.OpMode.PositionCorrection;
END_METHOD

END_FUNCTION_BLOCK

// ---- POUs/Prototypes/TcoDriveSimple/DriveState/TcoMovementState.TcPOU
FUNCTION_BLOCK INTERNAL TcoMovementState EXTENDS TcoCore.TcoState
VAR
    {attribute 'hide'}
    _axisRef : REFERENCE TO TcoAxisRef;
    {attribute 'hide'}
    _mcReset : Tc2_MC2.MC_Reset;
    {attribute 'hide'}
    _currentControlledTaskIdentity : ULINT;
END_VAR

PROPERTY DriveRef : REFERENCE TO TcoDriveSimple
GET
VAR
    _drive : ITcoDriveSimple := 0;
END_VAR
IF __QUERYINTERFACE(THIS^.Parent, _drive) THEN
    DriveRef REF= _drive.DriveRef;
END_IF
END_GET
END_PROPERTY

METHOD FB_init : BOOL
VAR_INPUT
    bInitRetains : BOOL; // if TRUE, the retain variables are initialized (warm start / cold start)
    bInCopyCode : BOOL; // if TRUE, the instance afterwards gets moved into the copy code (online change)
    ParentObject : ITcoObject;
    AutoRestoreMode : eRestoreMode;
END_VAR
END_METHOD

METHOD JogPreconditionsOk : BOOL
VAR_INPUT
    inObject : TcoCore.ITcoMomentaryTask;
    inParamsOK : BOOL;
END_VAR
VAR
    _controlledTask : TcoCore.ITcoMomentaryTask;
    _controlledTaskIdentity : ULINT;
END_VAR
JogPreconditionsOk := FALSE;

IF __QUERYINTERFACE(inObject, _controlledTask) THEN
    _controlledTaskIdentity := _controlledTask.Identity;
ELSE
    RETURN;
END_IF

IF NOT __ISVALIDREF(_axisRef) THEN
    IF __ISVALIDREF(DriveRef) THEN
        _axisRef REF= DriveRef.AxisRef;
    ELSE
        RETURN;
    END_IF
END_IF

IF THIS^.State = eTcoMovementState.WaitingForMovementTask THEN
    _mcReset(Axis := DriveRef.AxisRef, Execute := FALSE);

    IF _currentControlledTaskIdentity = 0 AND _controlledTaskIdentity <> 0 THEN
        _currentControlledTaskIdentity := _controlledTaskIdentity;

        IF THIS^.DriveRef._axisStatus.Error THEN
            THIS^.ChangeState(eTcoMovementState.Reset);
        ELSE
            THIS^.ChangeState(eTcoMovementState.Power);
        END_IF
    END_IF
END_IF

IF _currentControlledTaskIdentity = 0 OR _currentControlledTaskIdentity <> _controlledTaskIdentity THEN
    RETURN;
END_IF

IF THIS^.State = eTcoMovementState.Reset THEN
    _mcReset(Axis := DriveRef.AxisRef, Execute := TRUE);

    IF _mcReset.Done THEN
        _mcReset(Axis := DriveRef.AxisRef, Execute := FALSE);
        DriveRef.ClearError();
        DriveRef.RestoreTasks();
        _currentControlledTaskIdentity := _controlledTaskIdentity;
        THIS^.ChangeState(eTcoMovementState.Power);
    ELSIF _mcReset.Error THEN
        _mcReset(Axis := DriveRef.AxisRef, Execute := FALSE);
        THIS^.ChangeState(eTcoMovementState.Error);
    END_IF
END_IF

IF THIS^.State = eTcoMovementState.Power THEN
    IF NOT DriveRef._axisStatus.Disabled AND DriveRef._axisStatus.Operational THEN
        THIS^.ChangeState(eTcoMovementState.ParametersCheck);
    END_IF
END_IF

IF THIS^.State = eTcoMovementState.ParametersCheck THEN
    IF inParamsOK THEN
        THIS^.ChangeState(eTcoMovementState.Movement);
    END_IF
END_IF

IF THIS^.State = eTcoMovementState.Movement THEN
    JogPreconditionsOk := TRUE;
END_IF
END_METHOD

METHOD MovePreconditionsOk : BOOL
VAR_INPUT
    inObject : TcoCore.ITcoTask;
    inParamsOK : BOOL;
END_VAR
VAR
    _controlledTask : TcoCore.ITcoTask;
    _controlledTaskIdentity : ULINT;
END_VAR
MovePreconditionsOk := FALSE;

IF __QUERYINTERFACE(inObject, _controlledTask) THEN
    _controlledTaskIdentity := _controlledTask.Identity;
ELSE
    RETURN;
END_IF

IF NOT __ISVALIDREF(_axisRef) THEN
    IF __ISVALIDREF(DriveRef) THEN
        _axisRef REF= DriveRef.AxisRef;
    ELSE
        RETURN;
    END_IF
END_IF

IF THIS^.State = eTcoMovementState.WaitingForMovementTask THEN
    _mcReset(Axis := DriveRef.AxisRef, Execute := FALSE);

    IF _currentControlledTaskIdentity = 0 AND _controlledTaskIdentity <> 0 THEN
        _currentControlledTaskIdentity := _controlledTaskIdentity;

        IF THIS^.DriveRef._axisStatus.Error THEN
            THIS^.ChangeState(eTcoMovementState.Reset);
        ELSE
            THIS^.ChangeState(eTcoMovementState.Power);
        END_IF
    END_IF
END_IF

IF _currentControlledTaskIdentity = 0 OR _currentControlledTaskIdentity <> _controlledTaskIdentity THEN
    RETURN;
END_IF

IF THIS^.State = eTcoMovementState.Reset THEN
    _mcReset(Axis := DriveRef.AxisRef, Execute := TRUE);

    IF _mcReset.Done THEN
        _mcReset(Axis := DriveRef.AxisRef, Execute := FALSE);
        DriveRef.ClearError();
        DriveRef.RestoreTasks();
        _currentControlledTaskIdentity := _controlledTaskIdentity;
        THIS^.ChangeState(eTcoMovementState.Power);
        inObject.Invoke();
    ELSIF _mcReset.Error THEN
        _mcReset(Axis := DriveRef.AxisRef, Execute := FALSE);
        THIS^.ChangeState(eTcoMovementState.Error);
    END_IF
END_IF

IF THIS^.State = eTcoMovementState.Power THEN
    IF NOT DriveRef._axisStatus.Disabled AND DriveRef._axisStatus.Operational THEN
        THIS^.ChangeState(eTcoMovementState.ParametersCheck);
    END_IF
END_IF

IF THIS^.State = eTcoMovementState.ParametersCheck THEN
    IF inParamsOK THEN
        THIS^.ChangeState(eTcoMovementState.Movement);
    END_IF
END_IF

IF THIS^.State = eTcoMovementState.Movement THEN
    MovePreconditionsOk := TRUE;
END_IF
END_METHOD

METHOD Restore : ITcoRestorable
_currentControlledTaskIdentity := 0;
ChangeState(eTcoMovementState.WaitingForMovementTask);
END_METHOD

END_FUNCTION_BLOCK

// ---- POUs/Prototypes/TcoDriveSimple/Power.TcPOU
FUNCTION_BLOCK Power EXTENDS TcoCore.TcoObject IMPLEMENTS ITcoDriveSimple
VAR_INPUT
    inEnable : BOOL;
    inEnablePositive : BOOL;
    inEnableNegative : BOOL;
    inOverride : LREAL;
    inIsServiceMode : BOOL;
END_VAR
VAR
    {attribute addProperty Name "<#Power enable#>"}
    {attribute addProperty StateOnDesc "<#Enabled#>"}
    {attribute addProperty StateOffDesc "<#Disabled#>"}
    _driveEnableLocalTask : TcoCore.TcoToggleTask(THIS^, FALSE);
    {attribute addProperty Name "<#Enable positive#>"}
    {attribute addProperty StateOnDesc "<#Enabled#>"}
    {attribute addProperty StateOffDesc "<#Disabled#>"}
    _driveEnablePositiveLocalTask : TcoCore.TcoToggleTask(THIS^, FALSE);
    {attribute addProperty Name "<#Enable negative#>"}
    {attribute addProperty StateOnDesc "<#Enabled#>"}
    {attribute addProperty StateOffDesc "<#Disabled#>"}
    _driveEnableNegativeLocalTask : TcoCore.TcoToggleTask(THIS^, FALSE);
END_VAR
VAR
    {attribute 'hide'}
    _axisRef : REFERENCE TO TcoAxisRef;
    {attribute 'hide'}
    _mcPower : Tc2_MC2.MC_Power;
    {attribute addProperty Name "<#Drive power override#>"}
    {attribute addProperty StateOnDesc "<#Local control#>"}
    {attribute addProperty StateOffDesc "<#Global control#>"}
    _drivePowerOverrideTask : TcoCore.TcoToggleTask(THIS^, FALSE);
    {attribute 'hide'}
    _powerOverride : ePowerOverride;
    {attribute 'hide'}
    _powerOverridePV : ePowerOverride;
    {attribute addProperty Name "<#Override#>"}
    _override : LREAL;
    {attribute 'hide'}
    _enable : BOOL;
    {attribute 'hide'}
    _enablePositive : BOOL;
    {attribute 'hide'}
    _enableNegative : BOOL;
END_VAR

IF NOT __ISVALIDREF(_axisRef) THEN
    IF __ISVALIDREF(DriveRef) THEN
        _axisRef REF= DriveRef.AxisRef;
    ELSE
        RETURN;
    END_IF
END_IF

_drivePowerOverrideTask.Enabled := inIsServiceMode;
_drivePowerOverrideTask.Run();

IF _drivePowerOverrideTask.IsOff THEN
    _powerOverride := ePowerOverride.Global_control;
ELSE
    _powerOverride := ePowerOverride.Local_control;
END_IF;

_driveEnableLocalTask.Run();
_driveEnablePositiveLocalTask.Run();
_driveEnableNegativeLocalTask.Run();

//Take values from Global
IF _powerOverridePV = ePowerOverride.Global_control AND _powerOverride = ePowerOverride.Local_control THEN
    _override := inOverride;

    IF inEnable THEN
        _driveEnableLocalTask.On();
    ELSE
        _driveEnableLocalTask.Off();
    END_IF

    IF inEnablePositive THEN
        _driveEnablePositiveLocalTask.On();
    ELSE
        _driveEnablePositiveLocalTask.Off();
    END_IF

    IF inEnableNegative THEN
        _driveEnableNegativeLocalTask.On();
    ELSE
        _driveEnableNegativeLocalTask.Off();
    END_IF
END_IF

IF _powerOverridePV = ePowerOverride.Local_control AND _powerOverride = ePowerOverride.Global_control THEN
    IF inEnable THEN
        _driveEnableLocalTask.On();
    ELSE
        _driveEnableLocalTask.Off();
    END_IF

    IF inEnablePositive THEN
        _driveEnablePositiveLocalTask.On();
    ELSE
        _driveEnablePositiveLocalTask.Off();
    END_IF

    IF inEnableNegative THEN
        _driveEnableNegativeLocalTask.On();
    ELSE
        _driveEnableNegativeLocalTask.Off();
    END_IF

    _driveEnableLocalTask.Enabled := FALSE;
    _driveEnablePositiveLocalTask.Enabled := FALSE;
    _driveEnableNegativeLocalTask.Enabled := FALSE;
END_IF

_powerOverridePV := _powerOverride;

IF _powerOverride = ePowerOverride.Global_control THEN
    _mcPower(Axis := _axisRef,
        Enable := inEnable,
        Enable_Positive := inEnablePositive,
        Enable_Negative := inEnableNegative,
        Override := inOverride,
        BufferMode := Tc2_MC2.MC_BufferMode.MC_Aborting);
END_IF

IF _powerOverride = ePowerOverride.Local_control AND inIsServiceMode THEN
    _driveEnableLocalTask.Enabled := TRUE;
    _driveEnablePositiveLocalTask.Enabled := TRUE;
    _driveEnableNegativeLocalTask.Enabled := TRUE;

    _mcPower(Axis := _axisRef,
        Enable := _driveEnableLocalTask.State,
        Enable_Positive := _driveEnablePositiveLocalTask.State,
        Enable_Negative := _driveEnableNegativeLocalTask.State,
        Override := _override,
        BufferMode := Tc2_MC2.MC_BufferMode.MC_Aborting);
END_IF

IF NOT inIsServiceMode THEN
    IF _drivePowerOverrideTask.IsOn THEN
        _drivePowerOverrideTask.Off();
    END_IF

    _powerOverride := ePowerOverride.Global_control;
    _drivePowerOverrideTask.Enabled := FALSE;
    _driveEnableLocalTask.Enabled := FALSE;
    _driveEnablePositiveLocalTask.Enabled := FALSE;
    _driveEnableNegativeLocalTask.Enabled := FALSE;
END_IF

IF NOT _axisRef.Status.Error AND _mcPower.Error THEN
    DriveRef.SetErrorID(_mcPower.ErrorID);
END_IF

PROPERTY DriveRef : REFERENCE TO TcoDriveSimple
GET
VAR
    _drive : ITcoDriveSimple := 0;
END_VAR
IF __QUERYINTERFACE(THIS^.Parent, _drive) THEN
    DriveRef REF= _drive.DriveRef;
END_IF
END_GET
END_PROPERTY

METHOD FB_init : BOOL
VAR_INPUT
    bInitRetains : BOOL; // if TRUE, the retain variables are initialized (warm start / cold start)
    bInCopyCode : BOOL; // if TRUE, the instance afterwards gets moved into the copy code (online change)
    ParentObject : ITcoObject;
END_VAR
END_METHOD

END_FUNCTION_BLOCK

// ---- POUs/Prototypes/TcoDriveSimple/AxisTasks/ResetTask.TcPOU
FUNCTION_BLOCK ResetTask EXTENDS TcoCore.TcoTask IMPLEMENTS ITcoDriveSimple
VAR
    {attribute 'hide'}
    _axisRef : REFERENCE TO TcoAxisRef;
    {attribute 'hide'}
    _mcReset : Tc2_MC2.MC_Reset;
END_VAR

IF NOT __ISVALIDREF(_axisRef) THEN
    IF __ISVALIDREF(DriveRef) THEN
        _axisRef REF= DriveRef.AxisRef;
    ELSE
        RETURN;
    END_IF
END_IF

IF Execute() THEN
    _mcReset(Axis := _axisRef);
    DoneWhen(_mcReset.Done);
    ThrowWhen(_mcReset.Error);
END_IF

PROPERTY DriveRef : REFERENCE TO TcoDriveSimple
GET
VAR
    _drive : ITcoDriveSimple := 0;
END_VAR
IF __QUERYINTERFACE(THIS^.Parent, _drive) THEN
    DriveRef REF= _drive.DriveRef;
END_IF
END_GET
END_PROPERTY

METHOD PUBLIC FB_init : BOOL
VAR_INPUT
    bInitRetains : BOOL; // if TRUE, the retain variables are initialized (warm start / cold start)
    bInCopyCode : BOOL; // if TRUE, the instance afterwards gets moved into the copy code (online change)
    ParentObject : ITcoObject;
END_VAR
END_METHOD

(*~
    <docu>
        <summary>
            Executes when task reaches the ```Done``` state .
        </summary>
    </docu>
~*)
METHOD PROTECTED OnDone
DriveRef.RestoreTasks();
DriveRef.ClearError();
_mcReset(Axis := _axisRef, Execute := FALSE);
END_METHOD

(*~
    <docu>
        <summary>
            Executes when task reaches the ```Error``` state.
            <para>
                Do not confuse with <see cref="PlcDocu.TcoCore.TcoTask.WhileError()"/>, that is called cyclically until '''Error''' state is left.
            </para>
        </summary>
    </docu>
~*)
METHOD PROTECTED OnError
DriveRef.RestoreTasks();

IF NOT _axisRef.Status.Error THEN
    DriveRef.SetErrorID(DriveRef._resetTask._mcReset.ErrorID);
END_IF

_mcReset(Axis := _axisRef, Execute := FALSE);
END_METHOD

METHOD PROTECTED OnStart
DriveRef.ClearError();
_mcReset(Axis := _axisRef, Execute := TRUE);
END_METHOD

(*~
    <docu>
        <summary>
            Restores this instance to the Ready state. Can be called explicitly or from within one of the restore mechanisms.
            <para>
                See also <see cref="PlcDocu.TcoCore.TcoTask.AutoRestorable()"/>
            </para>
        </summary>
    </docu>
~*)
METHOD Restore : ITcoRestorable
SUPER^.Restore();
END_METHOD

(*~
    <docu>
        <summary>
            Executes until task is in ```Error``` state .
        </summary>
    </docu>
~*)
METHOD PROTECTED WhileError
IF NOT _axisRef.Status.Error THEN
    DriveRef.SetErrorID(DriveRef._resetTask._mcReset.ErrorID);
    _mcReset(Axis := _axisRef, Execute := FALSE);
END_IF
END_METHOD

END_FUNCTION_BLOCK

// ---- POUs/Prototypes/TcoDriveSimple/AxisTasks/SoEResetTask.TcPOU
FUNCTION_BLOCK SoEResetTask EXTENDS TcoCore.TcoTask IMPLEMENTS ITcoDriveSimple
VAR
    {attribute 'hide'}
    _axisRef : REFERENCE TO TcoAxisRef;
    {attribute 'hide'}
    _soEReset : Tc2_MC2_Drive.FB_SoEReset;
END_VAR

IF NOT __ISVALIDREF(_axisRef) THEN
    IF __ISVALIDREF(DriveRef) THEN
        _axisRef REF= DriveRef.AxisRef;
    ELSE
        RETURN;
    END_IF
END_IF

IF Execute() THEN
    _soEReset(Axis := _axisRef);
    DoneWhen(NOT _soEReset.Busy);
    ThrowWhen(_soEReset.Error);
END_IF

PROPERTY DriveRef : REFERENCE TO TcoDriveSimple
GET
VAR
    _drive : ITcoDriveSimple := 0;
END_VAR
IF __QUERYINTERFACE(THIS^.Parent, _drive) THEN
    DriveRef REF= _drive.DriveRef;
END_IF
END_GET
END_PROPERTY

METHOD PUBLIC FB_init : BOOL
VAR_INPUT
    bInitRetains : BOOL; // if TRUE, the retain variables are initialized (warm start / cold start)
    bInCopyCode : BOOL; // if TRUE, the instance afterwards gets moved into the copy code (online change)
    ParentObject : ITcoObject;
END_VAR
END_METHOD

(*~
    <docu>
        <summary>
            Executes when task reaches the ```Done``` state .
        </summary>
    </docu>
~*)
METHOD PROTECTED OnDone
_soEReset(NetId := _axisRef.ADS.NetId, Execute := FALSE, Axis := _axisRef);
THIS^.DriveRef._movementState.Restore();
END_METHOD

(*~
    <docu>
        <summary>
            Executes when task reaches the ```Error``` state.
            <para>
                Do not confuse with <see cref="PlcDocu.TcoCore.TcoTask.WhileError()"/>, that is called cyclically until '''Error''' state is left.
            </para>
        </summary>
    </docu>
~*)
METHOD PROTECTED OnError
THIS^.DriveRef._movementState.Restore();

IF NOT _axisRef.Status.Error THEN
    DriveRef.SetErrorID(DriveRef._soEResetTask._soEReset.AdsErrId);
END_IF

_soEReset(NetId := _axisRef.ADS.NetId, Execute := FALSE, Axis := _axisRef);
END_METHOD

METHOD PROTECTED OnStart
_soEReset(NetId := _axisRef.ADS.NetId, Execute := FALSE, Axis := _axisRef);
_soEReset(NetId := _axisRef.ADS.NetId, Execute := TRUE, Axis := _axisRef);
END_METHOD

(*~
    <docu>
        <summary>
            Restores this instance to the Ready state. Can be called explicitly or from within one of the restore mechanisms.
            <para>
                See also <see cref="PlcDocu.TcoCore.TcoTask.AutoRestorable()"/>
            </para>
        </summary>
    </docu>
~*)
METHOD Restore : ITcoRestorable
SUPER^.Restore();
END_METHOD

(*~
    <docu>
        <summary>
            Executes until task is in ```Error``` state .
        </summary>
    </docu>
~*)
METHOD PROTECTED WhileError
IF NOT _axisRef.Status.Error THEN
    DriveRef.SetErrorID(DriveRef._soEResetTask._soEReset.AdsErrId);
    _soEReset(Axis := _axisRef, Execute := FALSE);
END_IF
END_METHOD

END_FUNCTION_BLOCK

// ---- POUs/Prototypes/TcoDriveSimple/AxisTasks/SetPositionTask.TcPOU
FUNCTION_BLOCK SetPositionTask EXTENDS TcoCore.TcoTask IMPLEMENTS ITcoDriveSimple
VAR
    {attribute addProperty Name "<#Position#>"}
    _position : LREAL;
    {attribute addProperty Name "<#Mode#>"}
    _mode : eSetPositionMode;
END_VAR
VAR
    {attribute 'hide'}
    _axisRef : REFERENCE TO TcoAxisRef;
    {attribute 'hide'}
    _mcSetPosition : Tc2_MC2.MC_SetPosition;
    {attribute 'hide'}
    _mc_mode : BOOL;
    {attribute 'hide'}
    _message : STRING(125);
    {attribute 'hide'}
    _dummyPreconditionOK : BOOL;
END_VAR

IF NOT __ISVALIDREF(_axisRef) THEN
    IF __ISVALIDREF(DriveRef) THEN
        _axisRef REF= DriveRef.AxisRef;
    ELSE
        RETURN;
    END_IF
END_IF

IF Execute() THEN
    _dummyPreconditionOK := TRUE;

    IF NOT DriveRef._movementState.MovePreconditionsOk(THIS^, _dummyPreconditionOK) THEN
        Messenger.Error('To be implemented');
        RETURN;
    END_IF

    _mcSetPosition(Axis := _axisRef, Execute := TRUE, Position := _position);
    DoneWhen(_mcSetPosition.Done);
    ThrowWhen(_mcSetPosition.Error);
END_IF

PROPERTY DriveRef : REFERENCE TO TcoDriveSimple
GET
VAR
    _drive : ITcoDriveSimple := 0;
END_VAR
IF __QUERYINTERFACE(THIS^.Parent, _drive) THEN
    DriveRef REF= _drive.DriveRef;
END_IF
END_GET
END_PROPERTY

METHOD PUBLIC FB_init : BOOL
VAR_INPUT
    bInitRetains : BOOL; // if TRUE, the retain variables are initialized (warm start / cold start)
    bInCopyCode : BOOL; // if TRUE, the instance afterwards gets moved into the copy code (online change)
    ParentObject : ITcoObject;
END_VAR
END_METHOD

METHOD INTERNAL InvokeWithParams : ITcoTaskStatus
VAR_INPUT
    inPosition : LREAL;
    inMode : eSetPositionMode;
END_VAR
_position := inPosition;
_mode := inMode;
InvokeWithParams := THIS^.Invoke();
END_METHOD

(*~
    <docu>
        <summary>
            Executes when task reaches the ```Done``` state .
        </summary>
    </docu>
~*)
METHOD PROTECTED OnDone
_mcSetPosition(Axis := _axisRef, Execute := FALSE);
THIS^.DriveRef._movementState.Restore();
END_METHOD

(*~
    <docu>
        <summary>
            Executes when task reaches the ```Error``` state.
            <para>
                Do not confuse with <see cref="PlcDocu.TcoCore.TcoTask.WhileError()"/>, that is called cyclically until '''Error''' state is left.
            </para>
        </summary>
    </docu>
~*)
METHOD PROTECTED OnError
THIS^.DriveRef._movementState.Restore();

IF NOT _axisRef.Status.Error THEN
    DriveRef.SetErrorID(DriveRef._setPositionTask._mcSetPosition.ErrorID);
END_IF

_mcSetPosition(Axis := _axisRef, Execute := FALSE);
END_METHOD

METHOD PROTECTED OnStart
IF NOT Tco_TO_Tc2MC2_SetPositionMode(_mode, _mc_mode) THEN
    _message := Tc2_Standard.CONCAT('Unable to cast _mode variable of type TcoDrivesBeckhoff.eSetPositionMode (', TO_STRING(_mode));
    _message := Tc2_Standard.CONCAT(_message, ') to the type BOOL!!!');
    THIS^.Messenger.Post(_message, TcoCore.eMessageCategory.ProgrammingError);
    ThrowWhen(TRUE);
    RETURN;
END_IF

_mcSetPosition(Axis := _axisRef, Execute := FALSE);
END_METHOD

(*~
    <docu>
        <summary>
            Restores this instance to the Ready state. Can be called explicitly or from within one of the restore mechanisms.
            <para>
                See also <see cref="PlcDocu.TcoCore.TcoTask.AutoRestorable()"/>
            </para>
        </summary>
    </docu>
~*)
METHOD Restore : ITcoRestorable
SUPER^.Restore();
END_METHOD

(*~
    <docu>
        <summary>
            Executes until task is in ```Error``` state .
        </summary>
    </docu>
~*)
METHOD PROTECTED WhileError
IF NOT _axisRef.Status.Error THEN
    DriveRef.SetErrorID(DriveRef._setPositionTask._mcSetPosition.ErrorID);
    _mcSetPosition(Axis := _axisRef, Execute := FALSE);
END_IF
END_METHOD

END_FUNCTION_BLOCK

// ---- POUs/Prototypes/TcoDriveSimple/MotionTasks/HomeTask.TcPOU
FUNCTION_BLOCK HomeTask EXTENDS TcoCore.TcoTask IMPLEMENTS ITcoDriveSimple
VAR
    {attribute addProperty Name "<#Position#>"}
    _position : LREAL;
    {attribute addProperty Name "<#Mode#>"}
    _homingMode : eHomingMode;
    {attribute addProperty Name "<#Clear position lag#>"}
    _homingOptions_ClearPositionLag : BOOL;
    {attribute addProperty Name "<#Search direction#>"}
    _homingOptions_SearchDirection : eDirection;
    {attribute addProperty Name "<#Search velocity#>"}
    _homingOptions_SearchVelocity : LREAL;
    {attribute addProperty Name "<#Synchronization direction#>"}
    _homingOptions_SyncDirection : eDirection;
    {attribute addProperty Name "<#Synchronization velocity#>"}
    _homingOptions_SyncVelocity : LREAL;
    {attribute addProperty Name "<#Reference mode#>"}
    _homingOptions_ReferenceMode : eEncoderReferenceMode;
END_VAR
VAR
    {attribute 'hide'}
    _calibrationCam : BOOL;
    {attribute 'hide'}
    _axisRef : REFERENCE TO TcoAxisRef;
    {attribute 'hide'}
    _mcHome : Tc2_MC2.MC_Home;
    {attribute 'hide'}
    _mc_homingMode : Tc2_MC2.MC_HomingMode;
    {attribute 'hide'}
    _mc_homingOptions_SearchDirection : Tc2_MC2.MC_Direction;
    {attribute 'hide'}
    _mc_homingOptions_SyncDirection : Tc2_MC2.MC_Direction;
    {attribute 'hide'}
    _mc_homingOptions_ReferenceMode : Tc2_MC2.E_EncoderReferenceMode;
    {attribute 'hide'}
    _mc_homingOptions : Tc2_MC2.ST_HomingOptions;
    {attribute 'hide'}
    _message : STRING(125);
    {attribute 'hide'}
    _dummyPreconditionOK : BOOL;
END_VAR
VAR
    {attribute 'hide'}
    _sb : TcoCore.StringBuilder;
END_VAR

IF NOT __ISVALIDREF(_axisRef) THEN
    IF __ISVALIDREF(DriveRef) THEN
        _axisRef REF= DriveRef.AxisRef;
    ELSE
        RETURN;
    END_IF
END_IF

IF THIS^.Ready OR THIS^.Done THEN
    _mcHome(Axis := _axisRef, Execute := FALSE);
END_IF

IF Execute() THEN
    _dummyPreconditionOK := TRUE;

    IF NOT DriveRef._movementState.MovePreconditionsOk(THIS^, _dummyPreconditionOK) THEN
        Messenger.Error('To be implemented');
        RETURN;
    END_IF

    _calibrationCam := DriveRef.inCalibrationCam;

    _mcHome(Axis := _axisRef,
        Execute := NOT _mcHome.Busy,
        Position := _position,
        HomingMode := _mc_homingMode,
        BufferMode := Tc2_MC2.MC_Aborting,
        Options := _mc_homingOptions,
        bCalibrationCam := _calibrationCam,
        Done =>,
        Busy =>,
        Active =>,
        CommandAborted =>,
        Error =>,
        ErrorID =>);

    IF _mcHome.CommandAborted THEN
        THIS^.Abort();
    END_IF

    DoneWhen(_mcHome.Done);
    ThrowWhen(_mcHome.Error);
END_IF

IF (_mcHome.Error) THEN
    Messenger.Error(_sb.Clear()
            .Append('<#Homing error no #>')
            .Append(UDINT_TO_STRING(_mcHome.ErrorId))
            .Append(' |[[1]AdvancedDiagnosticMessage]|')
            .Append('.')
            .Append('For details see the service mode')
            .ToString());
END_IF;

PROPERTY DriveRef : REFERENCE TO TcoDriveSimple
GET
VAR
    _drive : ITcoDriveSimple := 0;
END_VAR
IF __QUERYINTERFACE(THIS^.Parent, _drive) THEN
    DriveRef REF= _drive.DriveRef;
END_IF
END_GET
END_PROPERTY

METHOD PUBLIC FB_init : BOOL
VAR_INPUT
    bInitRetains : BOOL; // if TRUE, the retain variables are initialized (warm start / cold start)
    bInCopyCode : BOOL; // if TRUE, the instance afterwards gets moved into the copy code (online change)
    ParentObject : ITcoObject;
END_VAR
END_METHOD

METHOD INTERNAL InvokeWithParams : ITcoTaskStatus
VAR_INPUT
    inPosition : LREAL;
    inHomingMode : eHomingMode;
    inClearPositionLag : BOOL;
    inSearchDirection : eDirection;
    inSearchVelocity : LREAL;
    inSyncDirection : eDirection;
    inSyncVelocity : LREAL;
    inReferenceMode : eEncoderReferenceMode;
END_VAR
_position := inPosition;
_homingMode := inHomingMode;
_homingOptions_ClearPositionLag := inClearPositionLag;
_homingOptions_SearchDirection := inSearchDirection;
_homingOptions_SearchVelocity := inSearchVelocity;
_homingOptions_SyncDirection := inSyncDirection;
_homingOptions_SyncVelocity := inSyncVelocity;
_homingOptions_ReferenceMode := inReferenceMode;
InvokeWithParams := THIS^.Invoke();
END_METHOD

(*~
    <docu>
        <summary>
            Executes when task is aborted.
        </summary>
    </docu>
~*)
METHOD PROTECTED OnAbort
IF NOT __ISVALIDREF(_axisRef) THEN
    IF __ISVALIDREF(DriveRef) THEN
        _axisRef REF= DriveRef.AxisRef;
    ELSE
        RETURN;
    END_IF
END_IF

THIS^.DriveRef.Stop(-1, -1);
_mcHome(Axis := _axisRef, Execute := FALSE);
THIS^.DriveRef._movementState.Restore();
END_METHOD

(*~
    <docu>
        <summary>
            Executes when task reaches the ```Done``` state .
        </summary>
    </docu>
~*)
METHOD PROTECTED OnDone
_mcHome(Axis := _axisRef, Execute := FALSE);
THIS^.DriveRef._movementState.Restore();
END_METHOD

(*~
    <docu>
        <summary>
            Executes when task reaches the ```Error``` state.
            <para>
                Do not confuse with <see cref="PlcDocu.TcoCore.TcoTask.WhileError()"/>, that is called cyclically until '''Error''' state is left.
            </para>
        </summary>
    </docu>
~*)
METHOD PROTECTED OnError
THIS^.DriveRef._movementState.Restore();

IF NOT _axisRef.Status.Error THEN
    DriveRef.SetErrorID(DriveRef._homeTask._mcHome.ErrorID);
END_IF

_mcHome(Axis := _axisRef, Execute := FALSE);
END_METHOD

